(* POU D2, LD *)
FUNCTION_BLOCK D2
VAR_INPUT
	pusk: BOOL;
	KUD2: BOOL;
	RMS2_2: BOOL;
	RD2: BOOL;
	TZD2:BOOL;
	avto: BOOL;
	GRIB: BOOL;
	stop_s: BOOL;
	ruchnoe: BOOL;
	pusk_LAN: BOOL;
	stop_LAN: BOOL;
	err: BOOL;
END_VAR
VAR_OUTPUT
	ready: BOOL;
	work: BOOL;
	KM2:BOOL;
	KM3:BOOL;
	stop_D3D4: BOOL;
	avar: BOOL;
END_VAR
VAR
	prom1: BOOL;
	start_KM3: TON;
	start_KM3_prom: TON;
	KM2_prom: BOOL;
	prom: BOOL;
	tof22: TOF;
END_VAR
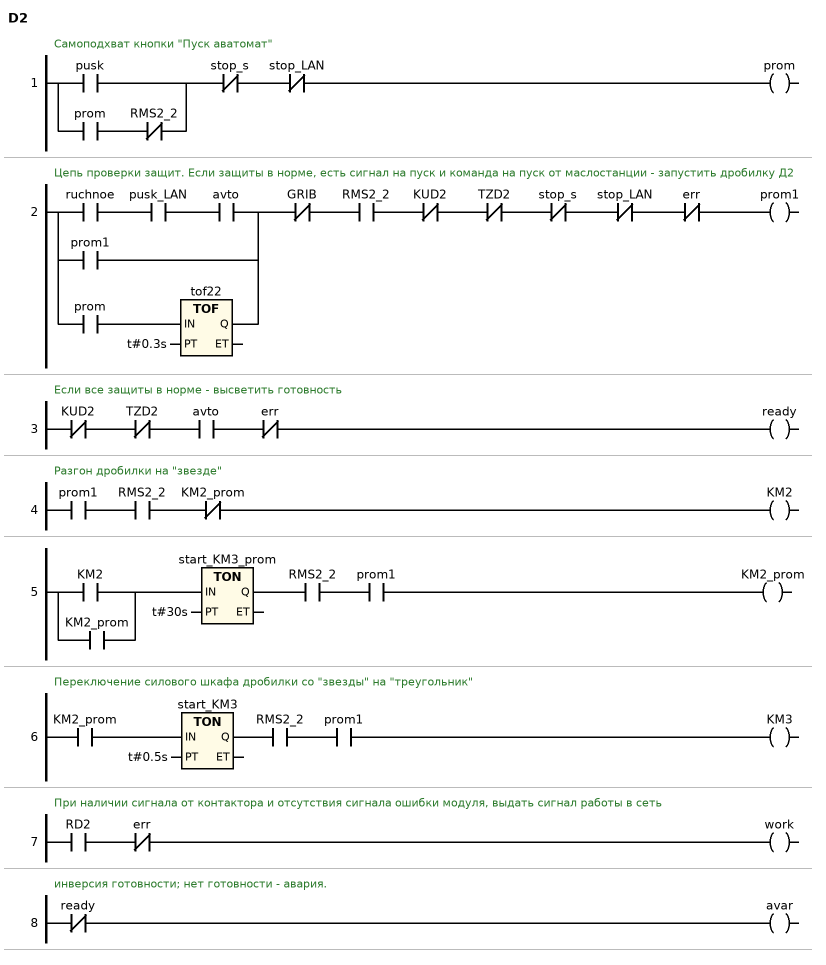
_LD_ (* Ladder Diagram *)
NETWORK 1 (* Самоподхват кнопки "Пуск аватомат" *)
	{ [pusk] | [prom] - [/RMS2_2] } - [/stop_s] - [/stop_LAN] --- (prom)
NETWORK 2 (* Цепь проверки защит. Если защиты в норме, есть сигнал на пуск и команда на пуск от маслостанции - запустить дробилку Д2 *)
	{ [ruchnoe] - [pusk_LAN] - [avto] | [prom1] | [prom] - tof22:TOF(IN: *, PT: t#0.3s) } - [/GRIB] - [RMS2_2] - [/KUD2] - [/TZD2] - [/stop_s] - [/stop_LAN] - [/err] --- (prom1)
NETWORK 3 (* Если все защиты в норме - высветить готовность *)
	[/KUD2] - [/TZD2] - [avto] - [/err] --- (ready)
NETWORK 4 (* Разгон дробилки на "звезде" *)
	[prom1] - [RMS2_2] - [/KM2_prom] --- (KM2)
NETWORK 5
	{ [KM2] | [KM2_prom] } - start_KM3_prom:TON(IN: *, PT: t#30s) - [RMS2_2] - [prom1] --- (KM2_prom)
NETWORK 6 (* Переключение силового шкафа дробилки со "звезды" на "треугольник" *)
	[KM2_prom] - start_KM3:TON(IN: *, PT: t#0.5s) - [RMS2_2] - [prom1] --- (KM3)
NETWORK 7 (* При наличии сигнала от контактора и отсутствия сигнала ошибки модуля, выдать сигнал работы в сеть *)
	[RD2] - [/err] --- (work)
NETWORK 8 (* инверсия готовности; нет готовности - авария. *)
	[/ready] --- (avar)
_END_LD_
(* the same logic as Structured Text *)
(* Network 1: Самоподхват кнопки "Пуск аватомат" *)
prom := (pusk OR prom AND NOT RMS2_2) AND NOT stop_s AND NOT stop_LAN;
(* Network 2: Цепь проверки защит. Если защиты в норме, есть сигнал на пуск и команда на пуск от маслостанции - запустить дробилку Д2 *)
tof22(IN := prom, PT := t#0.3s);
prom1 := (ruchnoe AND pusk_LAN AND avto OR prom1 OR tof22.Q) AND NOT GRIB AND RMS2_2 AND NOT KUD2 AND NOT TZD2 AND NOT stop_s AND NOT stop_LAN AND NOT err;
(* Network 3: Если все защиты в норме - высветить готовность *)
ready := NOT KUD2 AND NOT TZD2 AND avto AND NOT err;
(* Network 4: Разгон дробилки на "звезде" *)
KM2 := prom1 AND RMS2_2 AND NOT KM2_prom;
(* Network 5 *)
start_KM3_prom(IN := KM2 OR KM2_prom, PT := t#30s);
KM2_prom := start_KM3_prom.Q AND RMS2_2 AND prom1;
(* Network 6: Переключение силового шкафа дробилки со "звезды" на "треугольник" *)
start_KM3(IN := KM2_prom, PT := t#0.5s);
KM3 := start_KM3.Q AND RMS2_2 AND prom1;
(* Network 7: При наличии сигнала от контактора и отсутствия сигнала ошибки модуля, выдать сигнал работы в сеть *)
work := RD2 AND NOT err;
(* Network 8: инверсия готовности; нет готовности - авария. *)
avar := NOT ready;
END_FUNCTION_BLOCK

(* POU D3, LD *)
FUNCTION_BLOCK D3
VAR_INPUT
	pusk: BOOL;
	KU: BOOL;
	TZN: BOOL;
	KPM: BOOL;
	TZV: BOOL;

	KUD3: BOOL;
	TZD3: BOOL;
	RD3: BOOL;
	TM: WORD;
	RMS: BOOL;
	avto_in: BOOL;
	GRIB: BOOL;
	work_D2_D3: BOOL;
	stop_in: BOOL;
	ruchnoe: BOOL;
	pusk_LAN: BOOL;
	stop_LAN: BOOL;
	err: BOOL;
	UM: BOOL;
END_VAR

VAR_OUTPUT
	KM1: BOOL;
	KM2: BOOL;
	KM3: BOOL;
	ready: BOOL;
	nasos: BOOL;
	vent: BOOL;
	ten: BOOL;
	work: BOOL;
	avto:BOOL;
	avar: BOOL;
	stop_D3D4: BOOL;
	tm_ins: BOOL;
END_VAR

VAR
	prom1: BOOL;
	start_KM3: TON;
	KM2_prom: BOOL;
	start_KM3_prom: TON;
	run_pump: TON;
	prom2: BOOL;
	stop_D4: TON;
	stop_pump: TOF;
	tm_vent_ins: BOOL;
	tof1: TOF;
END_VAR
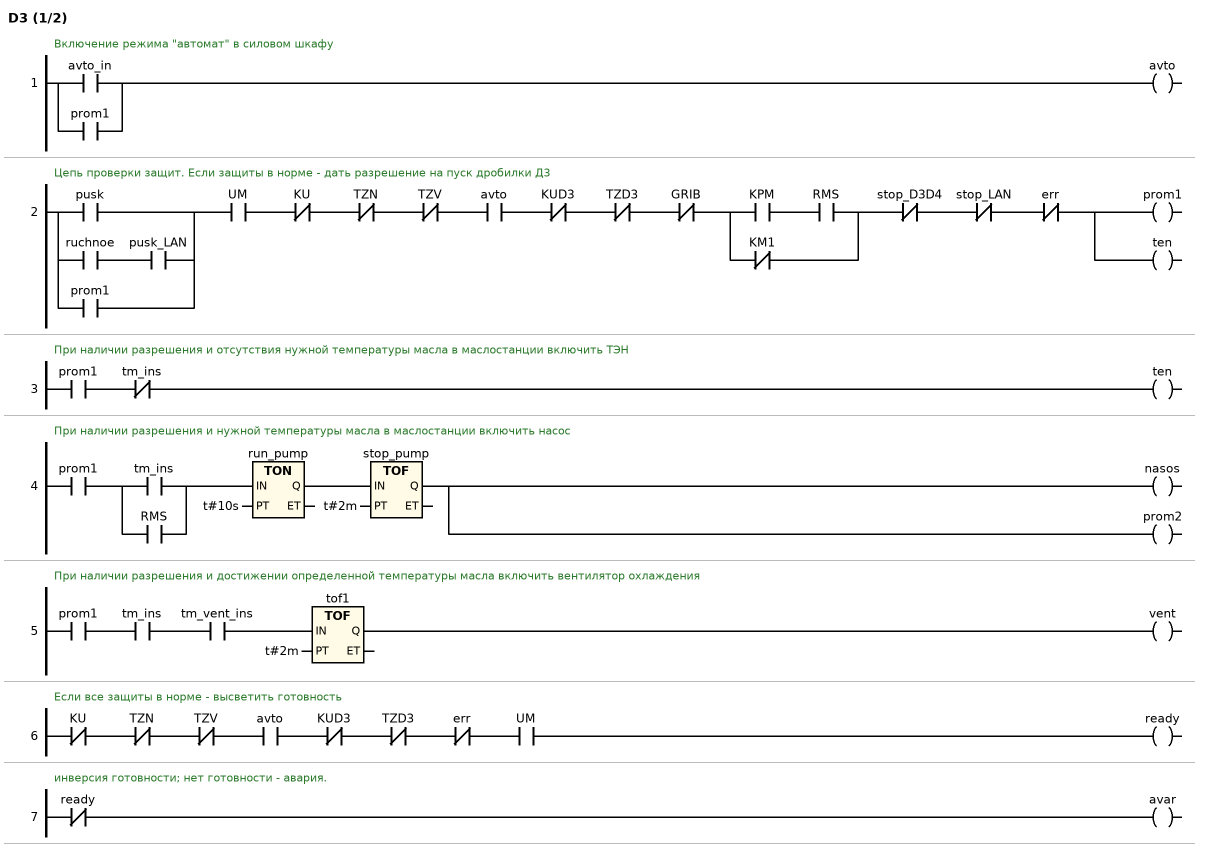
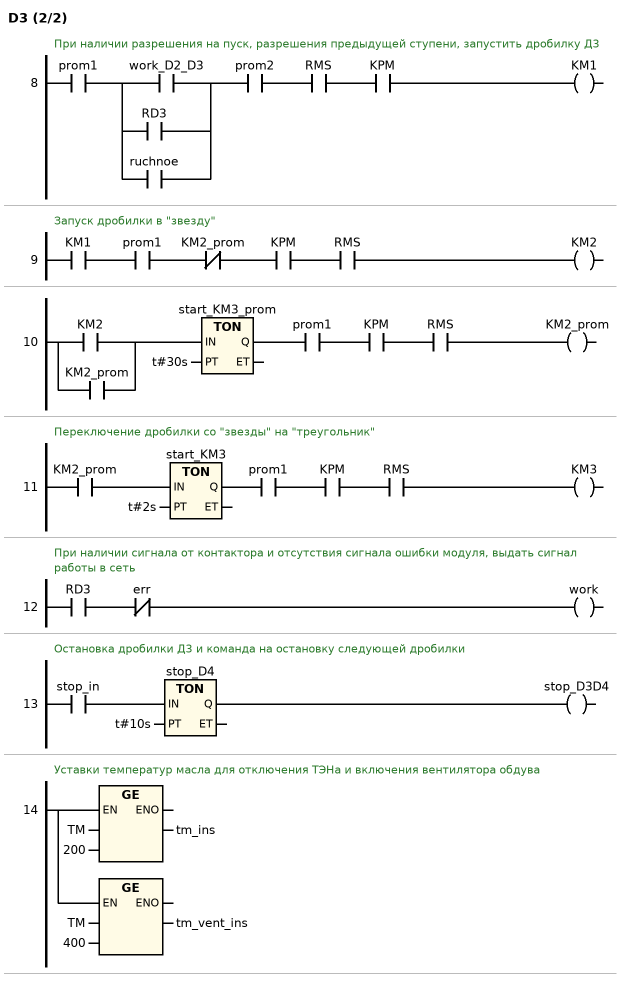
_LD_ (* Ladder Diagram *)
NETWORK 1 (* Включение режима "автомат" в силовом шкафу *)
	{ [avto_in] | [prom1] } --- (avto)
NETWORK 2 (* Цепь проверки защит. Если защиты в норме - дать разрешение на пуск дробилки Д3 *)
	{ [pusk] | [ruchnoe] - [pusk_LAN] | [prom1] } - [UM] - [/KU] - [/TZN] - [/TZV] - [avto] - [/KUD3] - [/TZD3] - [/GRIB] - { [KPM] - [RMS] | [/KM1] } - [/stop_D3D4] - [/stop_LAN] - [/err] --- (prom1) (ten)
NETWORK 3 (* При наличии разрешения и отсутствия нужной температуры масла в маслостанции включить ТЭН *)
	[prom1] - [/tm_ins] --- (ten)
NETWORK 4 (* При наличии разрешения и нужной температуры масла в маслостанции включить насос *)
	[prom1] - { [tm_ins] | [RMS] } - run_pump:TON(IN: *, PT: t#10s) - stop_pump:TOF(IN: *, PT: t#2m) --- (nasos) (prom2)
NETWORK 5 (* При наличии разрешения и достижении определенной температуры масла включить вентилятор охлаждения *)
	[prom1] - [tm_ins] - [tm_vent_ins] - tof1:TOF(IN: *, PT: t#2m) --- (vent)
NETWORK 6 (* Если все защиты в норме - высветить готовность *)
	[/KU] - [/TZN] - [/TZV] - [avto] - [/KUD3] - [/TZD3] - [/err] - [UM] --- (ready)
NETWORK 7 (* инверсия готовности; нет готовности - авария. *)
	[/ready] --- (avar)
NETWORK 8 (* При наличии разрешения на пуск, разрешения предыдущей ступени, запустить дробилку Д3 *)
	[prom1] - { [work_D2_D3] | [RD3] | [ruchnoe] } - [prom2] - [RMS] - [KPM] --- (KM1)
NETWORK 9 (* Запуск дробилки в "звезду" *)
	[KM1] - [prom1] - [/KM2_prom] - [KPM] - [RMS] --- (KM2)
NETWORK 10
	{ [KM2] | [KM2_prom] } - start_KM3_prom:TON(IN: *, PT: t#30s) - [prom1] - [KPM] - [RMS] --- (KM2_prom)
NETWORK 11 (* Переключение дробилки со "звезды" на "треугольник" *)
	[KM2_prom] - start_KM3:TON(IN: *, PT: t#2s) - [prom1] - [KPM] - [RMS] --- (KM3)
NETWORK 12 (* При наличии сигнала от контактора и отсутствия сигнала ошибки модуля, выдать сигнал работы в сеть *)
	[RD3] - [/err] --- (work)
NETWORK 13 (* Остановка дробилки Д3 и команда на остановку следующей дробилки *)
	[stop_in] - stop_D4:TON(IN: *, PT: t#10s) --- (stop_D3D4)
NETWORK 14 (* Уставки температур масла для отключения ТЭНа и включения вентилятора обдува *)
	*
		EN --- GE(TM, 200) => tm_ins
		EN --- GE(TM, 400) => tm_vent_ins
_END_LD_
(* the same logic as Structured Text *)
(* Network 1: Включение режима "автомат" в силовом шкафу *)
avto := avto_in OR prom1;
(* Network 2: Цепь проверки защит. Если защиты в норме - дать разрешение на пуск дробилки Д3 *)
prom1 := (pusk OR ruchnoe AND pusk_LAN OR prom1) AND UM AND NOT KU AND NOT TZN AND NOT TZV AND avto AND NOT KUD3 AND NOT TZD3 AND NOT GRIB AND (KPM AND RMS OR NOT KM1) AND NOT stop_D3D4 AND NOT stop_LAN AND NOT err;
ten := prom1;
(* Network 3: При наличии разрешения и отсутствия нужной температуры масла в маслостанции включить ТЭН *)
ten := prom1 AND NOT tm_ins;
(* Network 4: При наличии разрешения и нужной температуры масла в маслостанции включить насос *)
run_pump(IN := prom1 AND (tm_ins OR RMS), PT := t#10s);
stop_pump(IN := run_pump.Q, PT := t#2m);
nasos := stop_pump.Q;
prom2 := stop_pump.Q;
(* Network 5: При наличии разрешения и достижении определенной температуры масла включить вентилятор охлаждения *)
tof1(IN := prom1 AND tm_ins AND tm_vent_ins, PT := t#2m);
vent := tof1.Q;
(* Network 6: Если все защиты в норме - высветить готовность *)
ready := NOT KU AND NOT TZN AND NOT TZV AND avto AND NOT KUD3 AND NOT TZD3 AND NOT err AND UM;
(* Network 7: инверсия готовности; нет готовности - авария. *)
avar := NOT ready;
(* Network 8: При наличии разрешения на пуск, разрешения предыдущей ступени, запустить дробилку Д3 *)
KM1 := prom1 AND (work_D2_D3 OR RD3 OR ruchnoe) AND prom2 AND RMS AND KPM;
(* Network 9: Запуск дробилки в "звезду" *)
KM2 := KM1 AND prom1 AND NOT KM2_prom AND KPM AND RMS;
(* Network 10 *)
start_KM3_prom(IN := KM2 OR KM2_prom, PT := t#30s);
KM2_prom := start_KM3_prom.Q AND prom1 AND KPM AND RMS;
(* Network 11: Переключение дробилки со "звезды" на "треугольник" *)
start_KM3(IN := KM2_prom, PT := t#2s);
KM3 := start_KM3.Q AND prom1 AND KPM AND RMS;
(* Network 12: При наличии сигнала от контактора и отсутствия сигнала ошибки модуля, выдать сигнал работы в сеть *)
work := RD3 AND NOT err;
(* Network 13: Остановка дробилки Д3 и команда на остановку следующей дробилки *)
stop_D4(IN := stop_in, PT := t#10s);
stop_D3D4 := stop_D4.Q;
(* Network 14: Уставки температур масла для отключения ТЭНа и включения вентилятора обдува *)
tm_ins := TM >= 200;
tm_vent_ins := TM >= 400;
END_FUNCTION_BLOCK

(* POU D4, LD *)
FUNCTION_BLOCK D4
VAR_INPUT
	pusk: BOOL;
	KU: BOOL;
	TZN: BOOL;
	KPM: BOOL;
	TZV: BOOL;

	KUD3: BOOL;
	TZD3: BOOL;
	RD3: BOOL;
	TM: WORD;
	RMS: BOOL;
	avto_in: BOOL;
	GRIB: BOOL;
	work_D2_D3: BOOL;
	stop_in: BOOL;
	ruchnoe: BOOL;
	ins_0_40: BOOL;
	pusk_LAN: BOOL;
	stop_LAN: BOOL;
	err: BOOL;
	UM: BOOL;
END_VAR

VAR_OUTPUT
	KM1: BOOL;
	KM2: BOOL;
	KM3: BOOL;
	ready: BOOL;
	nasos: BOOL;
	vent: BOOL;
	ten: BOOL;
	work: BOOL;
	avto:BOOL;
	avar: BOOL;
	stop_D3D4: BOOL;
	tm_ins: BOOL;
END_VAR

VAR
	prom1: BOOL;
	start_KM3: TON;
	KM2_prom: BOOL;
	start_KM3_prom: TON;
	run_pump: TON;
	prom2: BOOL;
	stop_D4: TON;
	stop_pump: TOF;
	tm_vent_ins: BOOL;
	tof1: TOF;
END_VAR
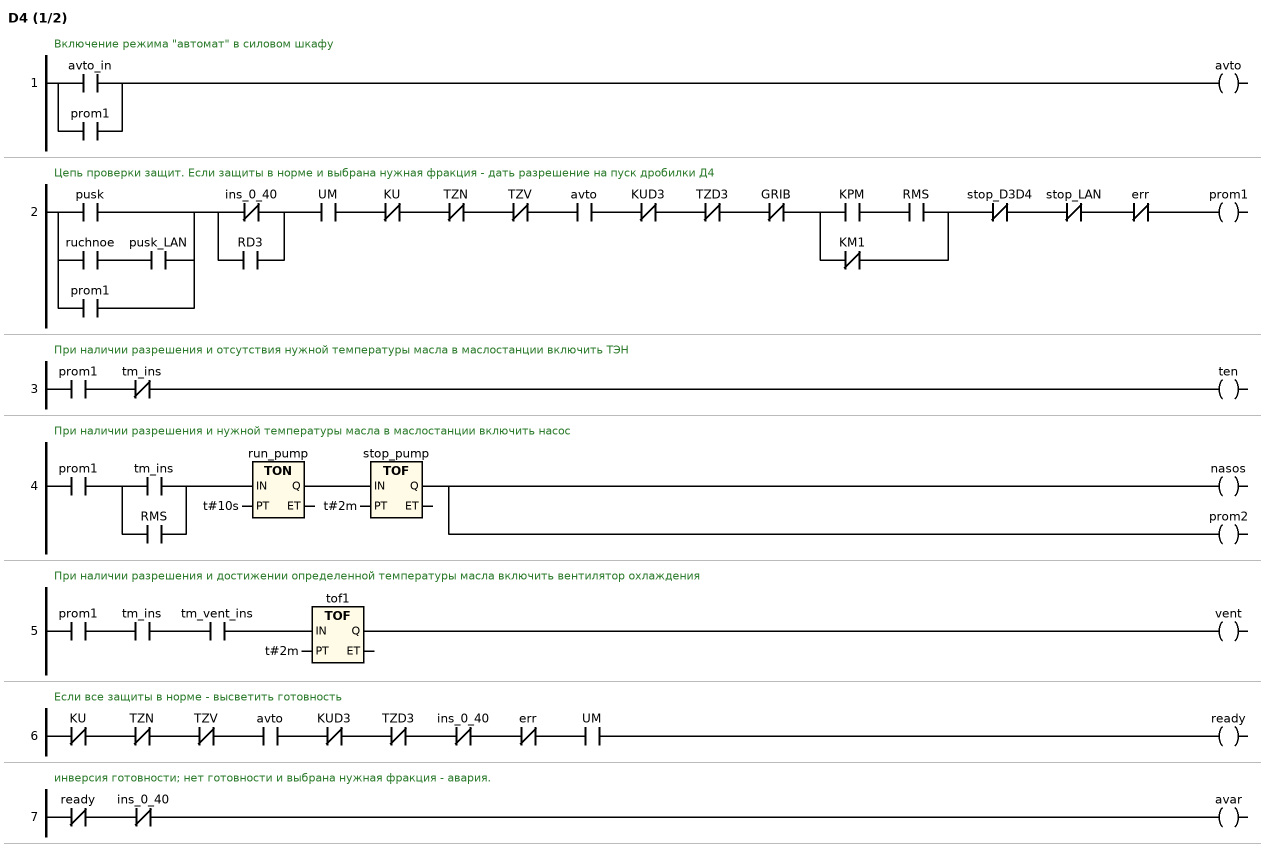
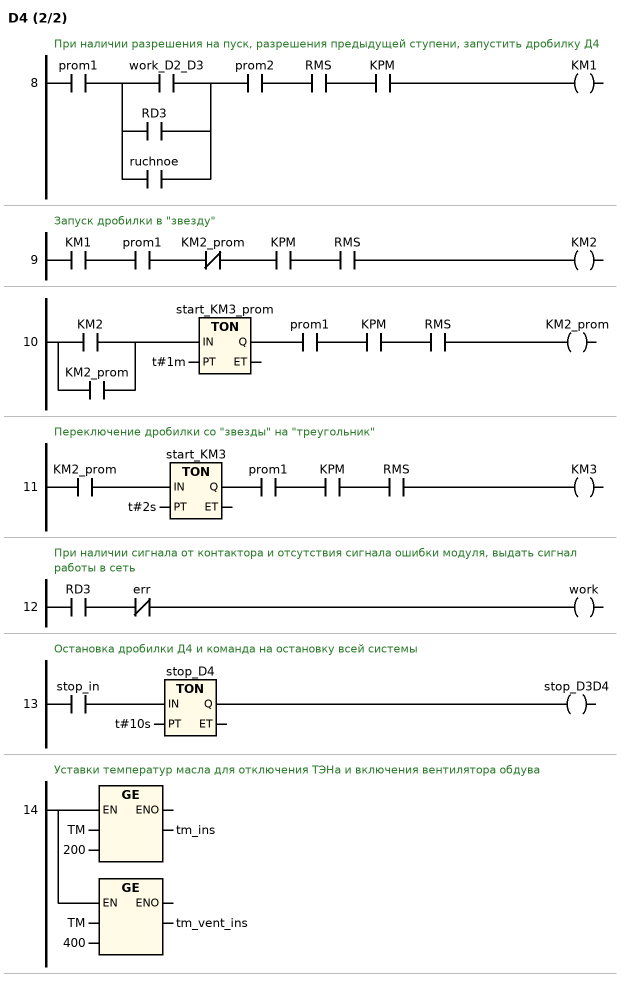
_LD_ (* Ladder Diagram *)
NETWORK 1 (* Включение режима "автомат" в силовом шкафу *)
	{ [avto_in] | [prom1] } --- (avto)
NETWORK 2 (* Цепь проверки защит. Если защиты в норме и выбрана нужная фракция - дать разрешение на пуск дробилки Д4 *)
	{ [pusk] | [ruchnoe] - [pusk_LAN] | [prom1] } - { [/ins_0_40] | [RD3] } - [UM] - [/KU] - [/TZN] - [/TZV] - [avto] - [/KUD3] - [/TZD3] - [/GRIB] - { [KPM] - [RMS] | [/KM1] } - [/stop_D3D4] - [/stop_LAN] - [/err] --- (prom1)
NETWORK 3 (* При наличии разрешения и отсутствия нужной температуры масла в маслостанции включить ТЭН *)
	[prom1] - [/tm_ins] --- (ten)
NETWORK 4 (* При наличии разрешения и нужной температуры масла в маслостанции включить насос *)
	[prom1] - { [tm_ins] | [RMS] } - run_pump:TON(IN: *, PT: t#10s) - stop_pump:TOF(IN: *, PT: t#2m) --- (nasos) (prom2)
NETWORK 5 (* При наличии разрешения и достижении определенной температуры масла включить вентилятор охлаждения *)
	[prom1] - [tm_ins] - [tm_vent_ins] - tof1:TOF(IN: *, PT: t#2m) --- (vent)
NETWORK 6 (* Если все защиты в норме - высветить готовность *)
	[/KU] - [/TZN] - [/TZV] - [avto] - [/KUD3] - [/TZD3] - [/ins_0_40] - [/err] - [UM] --- (ready)
NETWORK 7 (* инверсия готовности; нет готовности и выбрана нужная фракция - авария. *)
	[/ready] - [/ins_0_40] --- (avar)
NETWORK 8 (* При наличии разрешения на пуск, разрешения предыдущей ступени, запустить дробилку Д4 *)
	[prom1] - { [work_D2_D3] | [RD3] | [ruchnoe] } - [prom2] - [RMS] - [KPM] --- (KM1)
NETWORK 9 (* Запуск дробилки в "звезду" *)
	[KM1] - [prom1] - [/KM2_prom] - [KPM] - [RMS] --- (KM2)
NETWORK 10
	{ [KM2] | [KM2_prom] } - start_KM3_prom:TON(IN: *, PT: t#1m) - [prom1] - [KPM] - [RMS] --- (KM2_prom)
NETWORK 11 (* Переключение дробилки со "звезды" на "треугольник" *)
	[KM2_prom] - start_KM3:TON(IN: *, PT: t#2s) - [prom1] - [KPM] - [RMS] --- (KM3)
NETWORK 12 (* При наличии сигнала от контактора и отсутствия сигнала ошибки модуля, выдать сигнал работы в сеть *)
	[RD3] - [/err] --- (work)
NETWORK 13 (* Остановка дробилки Д4 и команда на остановку всей системы *)
	[stop_in] - stop_D4:TON(IN: *, PT: t#10s) --- (stop_D3D4)
NETWORK 14 (* Уставки температур масла для отключения ТЭНа и включения вентилятора обдува *)
	*
		EN --- GE(TM, 200) => tm_ins
		EN --- GE(TM, 400) => tm_vent_ins
_END_LD_
(* the same logic as Structured Text *)
(* Network 1: Включение режима "автомат" в силовом шкафу *)
avto := avto_in OR prom1;
(* Network 2: Цепь проверки защит. Если защиты в норме и выбрана нужная фракция - дать разрешение на пуск дробилки Д4 *)
prom1 := (pusk OR ruchnoe AND pusk_LAN OR prom1) AND (NOT ins_0_40 OR RD3) AND UM AND NOT KU AND NOT TZN AND NOT TZV AND avto AND NOT KUD3 AND NOT TZD3 AND NOT GRIB AND (KPM AND RMS OR NOT KM1) AND NOT stop_D3D4 AND NOT stop_LAN AND NOT err;
(* Network 3: При наличии разрешения и отсутствия нужной температуры масла в маслостанции включить ТЭН *)
ten := prom1 AND NOT tm_ins;
(* Network 4: При наличии разрешения и нужной температуры масла в маслостанции включить насос *)
run_pump(IN := prom1 AND (tm_ins OR RMS), PT := t#10s);
stop_pump(IN := run_pump.Q, PT := t#2m);
nasos := stop_pump.Q;
prom2 := stop_pump.Q;
(* Network 5: При наличии разрешения и достижении определенной температуры масла включить вентилятор охлаждения *)
tof1(IN := prom1 AND tm_ins AND tm_vent_ins, PT := t#2m);
vent := tof1.Q;
(* Network 6: Если все защиты в норме - высветить готовность *)
ready := NOT KU AND NOT TZN AND NOT TZV AND avto AND NOT KUD3 AND NOT TZD3 AND NOT ins_0_40 AND NOT err AND UM;
(* Network 7: инверсия готовности; нет готовности и выбрана нужная фракция - авария. *)
avar := NOT ready AND NOT ins_0_40;
(* Network 8: При наличии разрешения на пуск, разрешения предыдущей ступени, запустить дробилку Д4 *)
KM1 := prom1 AND (work_D2_D3 OR RD3 OR ruchnoe) AND prom2 AND RMS AND KPM;
(* Network 9: Запуск дробилки в "звезду" *)
KM2 := KM1 AND prom1 AND NOT KM2_prom AND KPM AND RMS;
(* Network 10 *)
start_KM3_prom(IN := KM2 OR KM2_prom, PT := t#1m);
KM2_prom := start_KM3_prom.Q AND prom1 AND KPM AND RMS;
(* Network 11: Переключение дробилки со "звезды" на "треугольник" *)
start_KM3(IN := KM2_prom, PT := t#2s);
KM3 := start_KM3.Q AND prom1 AND KPM AND RMS;
(* Network 12: При наличии сигнала от контактора и отсутствия сигнала ошибки модуля, выдать сигнал работы в сеть *)
work := RD3 AND NOT err;
(* Network 13: Остановка дробилки Д4 и команда на остановку всей системы *)
stop_D4(IN := stop_in, PT := t#10s);
stop_D3D4 := stop_D4.Q;
(* Network 14: Уставки температур масла для отключения ТЭНа и включения вентилятора обдува *)
tm_ins := TM >= 200;
tm_vent_ins := TM >= 400;
END_FUNCTION_BLOCK

(* POU LK1, LD *)
FUNCTION_BLOCK LK1 (*функциональный блок управления ленточными конвеерами 3, 5, 7, 8, 10-13*)
VAR_INPUT
	pusk: BOOL;
	avto:BOOL;
	KU: BOOL;
	TZ: BOOL;
	tros: BOOL;
	shod: BOOL;
	ogr: BOOL;
	VL:BOOL;
	P: BOOL;
	GRIB: BOOL;
	stop_s: BOOL;
	ruchnoe: BOOL;
	pusk_LAN: BOOL;
	stop_LAN: BOOL;
	err: BOOL;
	tros_self: BOOL;
	shod_self: BOOL;
	ogr_self: BOOL;
	pusk_sys_ins:BOOL;
END_VAR

VAR_OUTPUT
	KM:BOOL;
	ready: BOOL;
	work: BOOL;
	avar: BOOL;
	avar_vl: BOOL;
END_VAR

VAR
	prom1: BOOL;

	ftrig: F_TRIG;
	SR: SR;
END_VAR
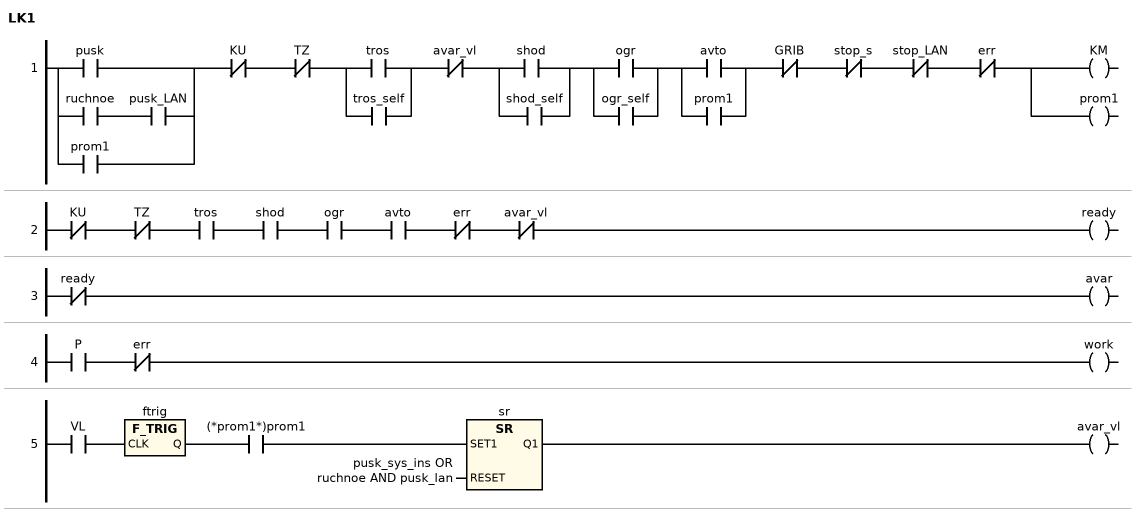
_LD_ (* Ladder Diagram *)
NETWORK 1
	{ [pusk] | [ruchnoe] - [pusk_LAN] | [prom1] } - [/KU] - [/TZ] - { [tros] | [tros_self] } - [/avar_vl] - { [shod] | [shod_self] } - { [ogr] | [ogr_self] } - { [avto] | [prom1] } - [/GRIB] - [/stop_s] - [/stop_LAN] - [/err] --- (KM) (prom1)
NETWORK 2
	[/KU] - [/TZ] - [tros] - [shod] - [ogr] - [avto] - [/err] - [/avar_vl] --- (ready)
NETWORK 3
	[/ready] --- (avar)
NETWORK 4
	[P] - [/err] --- (work)
NETWORK 5
	[VL] - ftrig:F_TRIG(CLK: *) - [(*prom1*)prom1] - sr:SR(SET1: *, RESET: pusk_sys_ins OR ruchnoe AND pusk_lan) --- (avar_vl)
_END_LD_
(* the same logic as Structured Text *)
(* Network 1 *)
KM := (pusk OR ruchnoe AND pusk_LAN OR prom1) AND NOT KU AND NOT TZ AND (tros OR tros_self) AND NOT avar_vl AND (shod OR shod_self) AND (ogr OR ogr_self) AND (avto OR prom1) AND NOT GRIB AND NOT stop_s AND NOT stop_LAN AND NOT err;
prom1 := KM;
(* Network 2 *)
ready := NOT KU AND NOT TZ AND tros AND shod AND ogr AND avto AND NOT err AND NOT avar_vl;
(* Network 3 *)
avar := NOT ready;
(* Network 4 *)
work := P AND NOT err;
(* Network 5 *)
ftrig(CLK := VL);
sr(SET1 := ftrig.Q AND ((*prom1*)prom1), RESET := pusk_sys_ins OR ruchnoe AND pusk_lan);
avar_vl := sr.Q1;
END_FUNCTION_BLOCK

(* POU counter, LD *)
FUNCTION_BLOCK counter  (* блок косвенного подсчёта скорости, исходя из приходящего количества импульсов*)
VAR_INPUT
	Vl: WORD;
	work: BOOL;
	in_time: WORD;
END_VAR
VAR_OUTPUT
	out_Vl: BOOL;
END_VAR
VAR
	vl_ins: WORD;
	vl_eq: BOOL;
	ton1: TOF;
	blink1: BLINK;
	tp1: TP;
	vl_sub: WORD;
	ins_time: WORD;
	time_read: TIME;
END_VAR
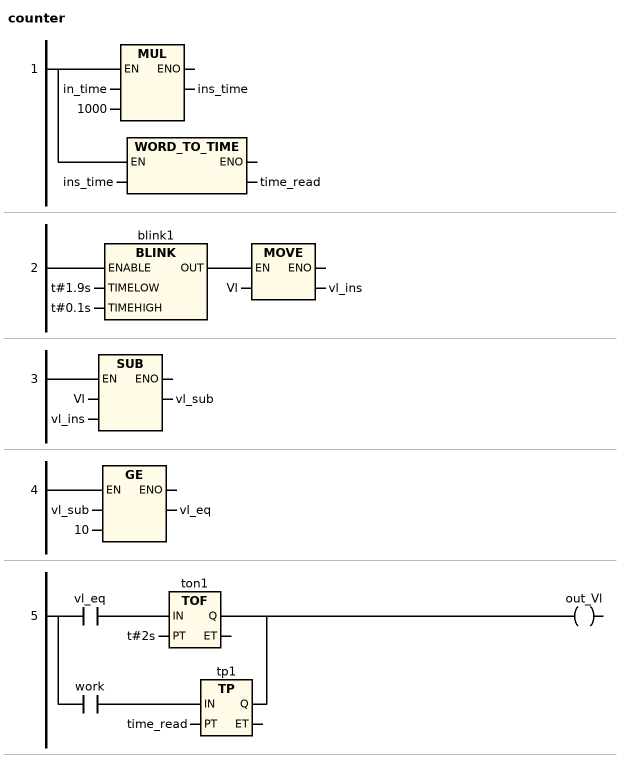
_LD_ (* Ladder Diagram *)
NETWORK 1
	*
		EN --- MUL(in_time, 1000) => ins_time
		EN --- WORD_TO_TIME(ins_time) => time_read
NETWORK 2
	blink1:BLINK(ENABLE: *, TIMELOW: t#1.9s, TIMEHIGH: t#0.1s)
		EN --- MOVE(Vl) => vl_ins
NETWORK 3
	*
		EN --- SUB(Vl, vl_ins) => vl_sub
NETWORK 4
	*
		EN --- GE(vl_sub, 10) => vl_eq
NETWORK 5
	{ [vl_eq] - ton1:TOF(IN: *, PT: t#2s) | [work] - tp1:TP(IN: *, PT: time_read) } --- (out_Vl)
_END_LD_
(* the same logic as Structured Text *)
(* Network 1 *)
ins_time := in_time * 1000;
time_read := WORD_TO_TIME(ins_time);
(* Network 2 *)
blink1(ENABLE := TRUE, TIMELOW := t#1.9s, TIMEHIGH := t#0.1s);
IF blink1.OUT THEN
	vl_ins := Vl;
END_IF;
(* Network 3 *)
vl_sub := Vl - vl_ins;
(* Network 4 *)
vl_eq := vl_sub >= 10;
(* Network 5 *)
ton1(IN := vl_eq, PT := t#2s);
tp1(IN := work, PT := time_read);
out_Vl := ton1.Q OR tp1.Q;
END_FUNCTION_BLOCK

(* POU LK12, LD *)
FUNCTION_BLOCK LK12 (*функциональный блок управления ленточными конвеерами 3, 5, 7, 8, 10-13*)
VAR_INPUT
	avto:BOOL;
	KU: BOOL;
	TZ: BOOL;
	tros: BOOL;
	shod: BOOL;
	ogr: BOOL;
	VL:BOOL;
	P: BOOL;
	GRIB: BOOL;
	stop_s: BOOL;
	ruchnoe: BOOL;
	pusk_LAN: BOOL;
	stop_LAN: BOOL;
	err: BOOL;
	tros_self: BOOL;
	shod_self: BOOL;
	ogr_self: BOOL;
	pusk_sys_ins:BOOL;
END_VAR

VAR_OUTPUT
	KM:BOOL;
	ready: BOOL;
	work: BOOL;
	avar: BOOL;
	avar_vl: BOOL;
END_VAR

VAR
	prom1: BOOL;

	ftrig: F_TRIG;
	SR: SR;
END_VAR
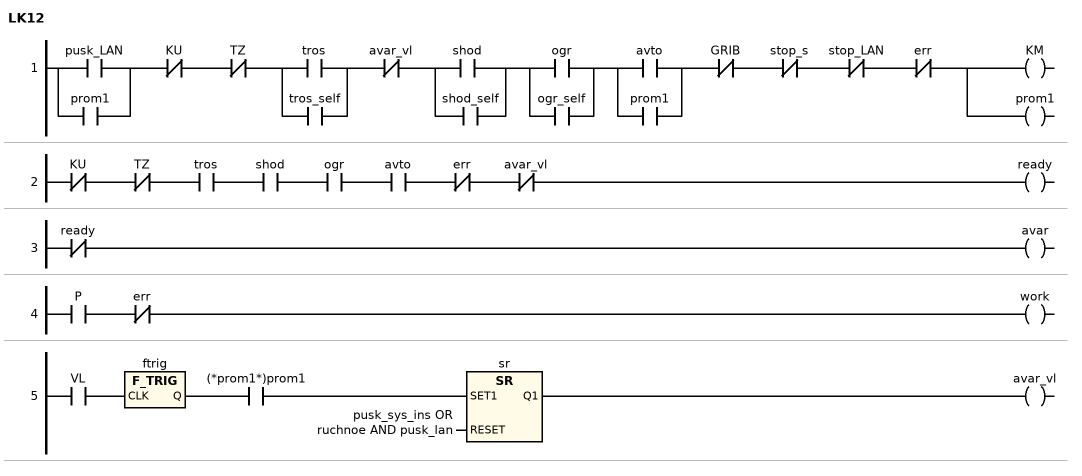
_LD_ (* Ladder Diagram *)
NETWORK 1
	{ [pusk_LAN] | [prom1] } - [/KU] - [/TZ] - { [tros] | [tros_self] } - [/avar_vl] - { [shod] | [shod_self] } - { [ogr] | [ogr_self] } - { [avto] | [prom1] } - [/GRIB] - [/stop_s] - [/stop_LAN] - [/err] --- (KM) (prom1)
NETWORK 2
	[/KU] - [/TZ] - [tros] - [shod] - [ogr] - [avto] - [/err] - [/avar_vl] --- (ready)
NETWORK 3
	[/ready] --- (avar)
NETWORK 4
	[P] - [/err] --- (work)
NETWORK 5
	[VL] - ftrig:F_TRIG(CLK: *) - [(*prom1*)prom1] - sr:SR(SET1: *, RESET: pusk_sys_ins OR ruchnoe AND pusk_lan) --- (avar_vl)
_END_LD_
(* the same logic as Structured Text *)
(* Network 1 *)
KM := (pusk_LAN OR prom1) AND NOT KU AND NOT TZ AND (tros OR tros_self) AND NOT avar_vl AND (shod OR shod_self) AND (ogr OR ogr_self) AND (avto OR prom1) AND NOT GRIB AND NOT stop_s AND NOT stop_LAN AND NOT err;
prom1 := KM;
(* Network 2 *)
ready := NOT KU AND NOT TZ AND tros AND shod AND ogr AND avto AND NOT err AND NOT avar_vl;
(* Network 3 *)
avar := NOT ready;
(* Network 4 *)
work := P AND NOT err;
(* Network 5 *)
ftrig(CLK := VL);
sr(SET1 := ftrig.Q AND ((*prom1*)prom1), RESET := pusk_sys_ins OR ruchnoe AND pusk_lan);
avar_vl := sr.Q1;
END_FUNCTION_BLOCK

(* POU LK12_modern, LD *)
FUNCTION_BLOCK LK12_modern (*функциональный блок управления ленточными конвеерами 12*)
VAR_INPUT
	pusk: BOOL;
	avto:BOOL;
	KU: BOOL;
	TZ: BOOL;
	tros: BOOL;
	shod: BOOL;
	ogr: BOOL;
	VL:BOOL;
	P: BOOL;
	GRIB: BOOL;
	stop_s: BOOL;
	ruchnoe: BOOL;
	pusk_LAN: BOOL;
	stop_LAN: BOOL;
	err: BOOL;
	tros_self: BOOL;
	shod_self: BOOL;
	ogr_self: BOOL;
	pusk_sys_ins:BOOL;
	switcher_in: WORD;
	current_value_lk12_in: BOOL;
END_VAR

VAR_OUTPUT
	KM:BOOL;
	ready: BOOL;
	work: BOOL;
	avar: BOOL;
	avar_vl: BOOL;
	current_value_lk12_out: BOOL;
END_VAR

VAR
	prom1: BOOL;

	ftrig: F_TRIG;
	SR: SR;
	switcher_in_bool: BOOL;
	lk12_trig: lk12_trig;
END_VAR
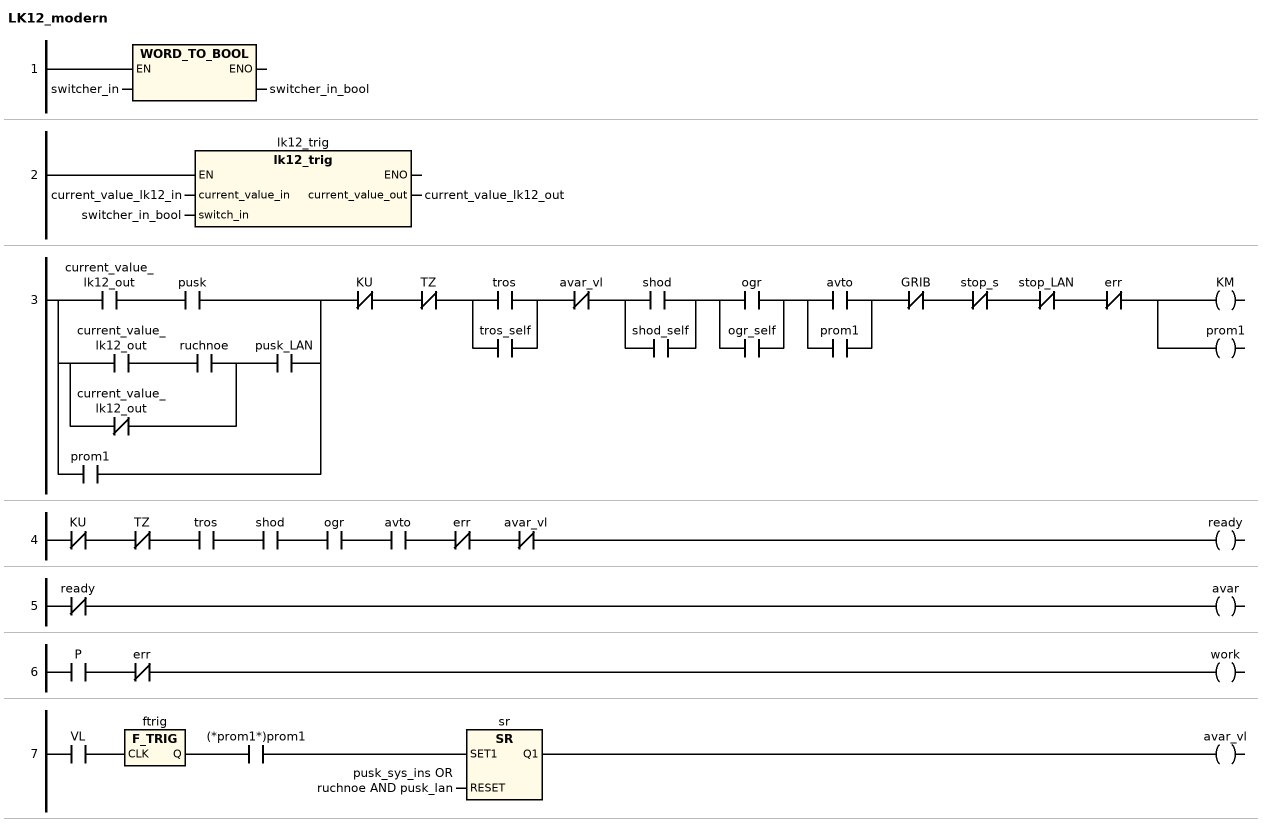
_LD_ (* Ladder Diagram *)
NETWORK 1
	*
		EN --- WORD_TO_BOOL(switcher_in) => switcher_in_bool
NETWORK 2
	*
		EN --- lk12_trig:lk12_trig(current_value_in: current_value_lk12_in, switch_in: switcher_in_bool) => current_value_lk12_out
NETWORK 3
	{ [current_value_lk12_out] - [pusk] | { [current_value_lk12_out] - [ruchnoe] | [/current_value_lk12_out] } - [pusk_LAN] | [prom1] } - [/KU] - [/TZ] - { [tros] | [tros_self] } - [/avar_vl] - { [shod] | [shod_self] } - { [ogr] | [ogr_self] } - { [avto] | [prom1] } - [/GRIB] - [/stop_s] - [/stop_LAN] - [/err] --- (KM) (prom1)
NETWORK 4
	[/KU] - [/TZ] - [tros] - [shod] - [ogr] - [avto] - [/err] - [/avar_vl] --- (ready)
NETWORK 5
	[/ready] --- (avar)
NETWORK 6
	[P] - [/err] --- (work)
NETWORK 7
	[VL] - ftrig:F_TRIG(CLK: *) - [(*prom1*)prom1] - sr:SR(SET1: *, RESET: pusk_sys_ins OR ruchnoe AND pusk_lan) --- (avar_vl)
_END_LD_
(* the same logic as Structured Text *)
(* Network 1 *)
switcher_in_bool := WORD_TO_BOOL(switcher_in);
(* Network 2 *)
lk12_trig(current_value_in := current_value_lk12_in, switch_in := switcher_in_bool);
current_value_lk12_out := lk12_trig.current_value_out;
(* Network 3 *)
KM := (current_value_lk12_out AND pusk OR (current_value_lk12_out AND ruchnoe OR NOT current_value_lk12_out) AND pusk_LAN OR prom1) AND NOT KU AND NOT TZ AND (tros OR tros_self) AND NOT avar_vl AND (shod OR shod_self) AND (ogr OR ogr_self) AND (avto OR prom1) AND NOT GRIB AND NOT stop_s AND NOT stop_LAN AND NOT err;
prom1 := KM;
(* Network 4 *)
ready := NOT KU AND NOT TZ AND tros AND shod AND ogr AND avto AND NOT err AND NOT avar_vl;
(* Network 5 *)
avar := NOT ready;
(* Network 6 *)
work := P AND NOT err;
(* Network 7 *)
ftrig(CLK := VL);
sr(SET1 := ftrig.Q AND ((*prom1*)prom1), RESET := pusk_sys_ins OR ruchnoe AND pusk_lan);
avar_vl := sr.Q1;
END_FUNCTION_BLOCK

(* POU lk12_trig, ST *)
FUNCTION_BLOCK lk12_trig
VAR_INPUT
	current_value_in: BOOL;
	switch_in: BOOL;
END_VAR
VAR_OUTPUT
	current_value_out: BOOL;
END_VAR
VAR
	rtrig : R_TRIG;
	rtrigQ: BOOL;
END_VAR
rtrig(CLK := switch_in);
rtrigQ := rtrig.Q;

IF current_value_in = TRUE AND rtrigQ = TRUE
THEN
current_value_out := FALSE;
ELSIF current_value_in = FALSE AND rtrigQ = TRUE
THEN
current_value_out := TRUE;
END_IF
END_FUNCTION_BLOCK

(* POU Grohot, LD *)
FUNCTION_BLOCK Grohot
VAR_INPUT
	pusk: BOOL;
	avto: BOOL;
	KU: BOOL;
	TZ: BOOL;
	P:BOOL;
	STOP: BOOL;
	GRIB: BOOL;
	stop_s: BOOL;
	ruchnoe: BOOL;
	pusk_LAN: BOOL;
	stop_LAN: BOOL;
	err: BOOL;
END_VAR

VAR_OUTPUT
	KM: BOOL;
	ready: BOOL;
	work: BOOL;
	avar: BOOL;
END_VAR

VAR
	prom1: BOOL;
END_VAR
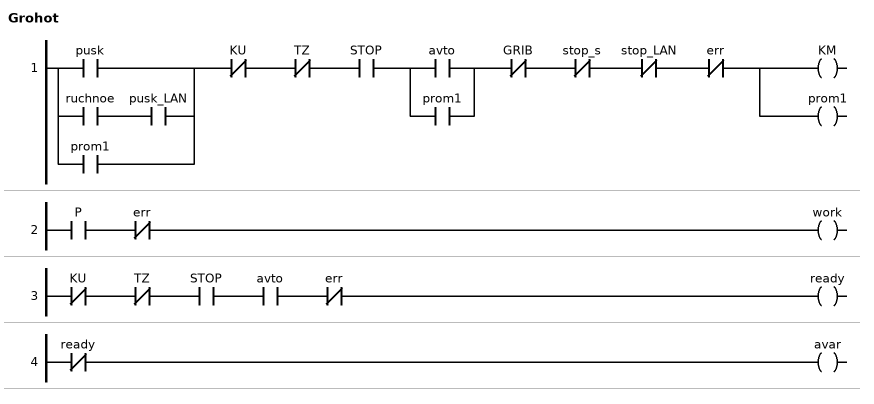
_LD_ (* Ladder Diagram *)
NETWORK 1
	{ [pusk] | [ruchnoe] - [pusk_LAN] | [prom1] } - [/KU] - [/TZ] - [STOP] - { [avto] | [prom1] } - [/GRIB] - [/stop_s] - [/stop_LAN] - [/err] --- (KM) (prom1)
NETWORK 2
	[P] - [/err] --- (work)
NETWORK 3
	[/KU] - [/TZ] - [STOP] - [avto] - [/err] --- (ready)
NETWORK 4
	[/ready] --- (avar)
_END_LD_
(* the same logic as Structured Text *)
(* Network 1 *)
KM := (pusk OR ruchnoe AND pusk_LAN OR prom1) AND NOT KU AND NOT TZ AND STOP AND (avto OR prom1) AND NOT GRIB AND NOT stop_s AND NOT stop_LAN AND NOT err;
prom1 := KM;
(* Network 2 *)
work := P AND NOT err;
(* Network 3 *)
ready := NOT KU AND NOT TZ AND STOP AND avto AND NOT err;
(* Network 4 *)
avar := NOT ready;
END_FUNCTION_BLOCK

(* POU LK3, LD *)
FUNCTION_BLOCK LK3  (*Ленточный конвееры 6*)
VAR_INPUT
	pusk: BOOL;
	avto:BOOL;
	KU: BOOL;
	TZ: BOOL;
	tros: BOOL;
	shod: BOOL;
	ogr: BOOL;
	VL:BOOL;
	P:BOOL;
	in_020: BOOL;
	stop_s: BOOL;
	GRIB: BOOL;
	ruchnoe: BOOL;
	pusk_LAN: BOOL;
	stop_LAN: BOOL;
	err: BOOL;
	tros_self: BOOL;
	shod_self: BOOL;
	ogr_self: BOOL;
	pusk_sys_ins:BOOL;
END_VAR

VAR_OUTPUT
	KM: BOOL;
	ready: BOOL;
	work: BOOL;
	avar: BOOL;
	avar_vl: BOOL;
END_VAR

VAR
	prom1: BOOL;

	ftrig: F_TRIG;
	SR: SR;
END_VAR
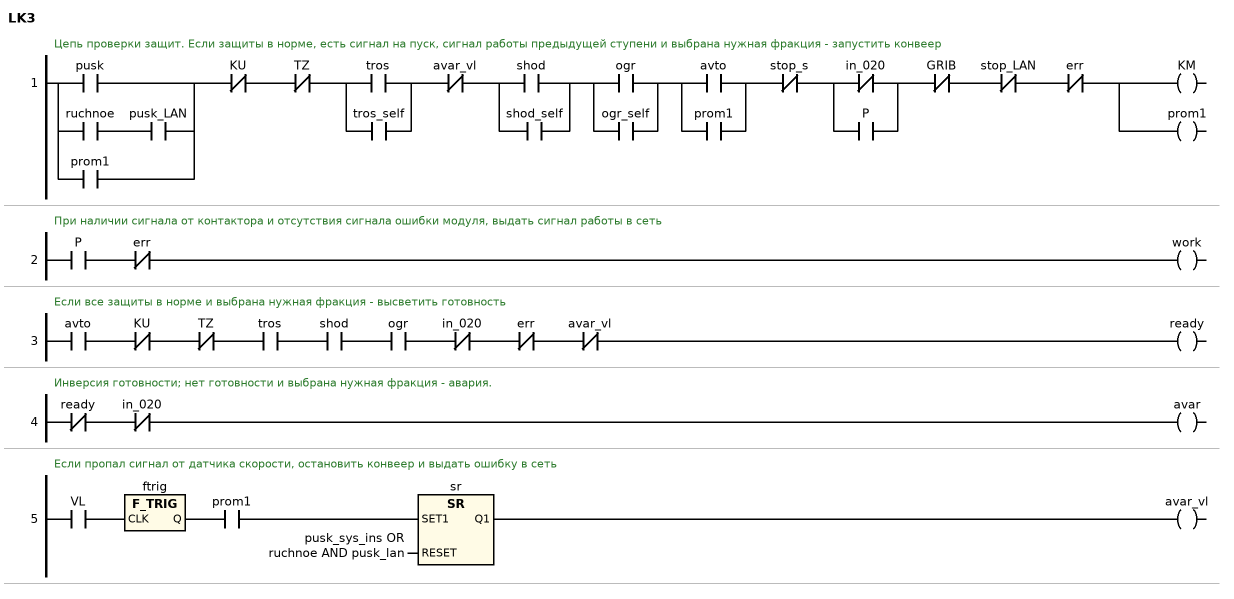
_LD_ (* Ladder Diagram *)
NETWORK 1 (* Цепь проверки защит. Если защиты в норме, есть сигнал на пуск, сигнал работы предыдущей ступени и выбрана нужная фракция - запустить конвеер *)
	{ [pusk] | [ruchnoe] - [pusk_LAN] | [prom1] } - [/KU] - [/TZ] - { [tros] | [tros_self] } - [/avar_vl] - { [shod] | [shod_self] } - { [ogr] | [ogr_self] } - { [avto] | [prom1] } - [/stop_s] - { [/in_020] | [P] } - [/GRIB] - [/stop_LAN] - [/err] --- (KM) (prom1)
NETWORK 2 (* При наличии сигнала от контактора и отсутствия сигнала ошибки модуля, выдать сигнал работы в сеть *)
	[P] - [/err] --- (work)
NETWORK 3 (* Если все защиты в норме и выбрана нужная фракция - высветить готовность *)
	[avto] - [/KU] - [/TZ] - [tros] - [shod] - [ogr] - [/in_020] - [/err] - [/avar_vl] --- (ready)
NETWORK 4 (* Инверсия готовности; нет готовности и выбрана нужная фракция - авария. *)
	[/ready] - [/in_020] --- (avar)
NETWORK 5 (* Если пропал сигнал от датчика скорости, остановить конвеер и выдать ошибку в сеть *)
	[VL] - ftrig:F_TRIG(CLK: *) - [prom1] - sr:SR(SET1: *, RESET: pusk_sys_ins OR ruchnoe AND pusk_lan) --- (avar_vl)
_END_LD_
(* the same logic as Structured Text *)
(* Network 1: Цепь проверки защит. Если защиты в норме, есть сигнал на пуск, сигнал работы предыдущей ступени и выбрана нужная фракция - запустить конвеер *)
KM := (pusk OR ruchnoe AND pusk_LAN OR prom1) AND NOT KU AND NOT TZ AND (tros OR tros_self) AND NOT avar_vl AND (shod OR shod_self) AND (ogr OR ogr_self) AND (avto OR prom1) AND NOT stop_s AND (NOT in_020 OR P) AND NOT GRIB AND NOT stop_LAN AND NOT err;
prom1 := KM;
(* Network 2: При наличии сигнала от контактора и отсутствия сигнала ошибки модуля, выдать сигнал работы в сеть *)
work := P AND NOT err;
(* Network 3: Если все защиты в норме и выбрана нужная фракция - высветить готовность *)
ready := avto AND NOT KU AND NOT TZ AND tros AND shod AND ogr AND NOT in_020 AND NOT err AND NOT avar_vl;
(* Network 4: Инверсия готовности; нет готовности и выбрана нужная фракция - авария. *)
avar := NOT ready AND NOT in_020;
(* Network 5: Если пропал сигнал от датчика скорости, остановить конвеер и выдать ошибку в сеть *)
ftrig(CLK := VL);
sr(SET1 := ftrig.Q AND prom1, RESET := pusk_sys_ins OR ruchnoe AND pusk_lan);
avar_vl := sr.Q1;
END_FUNCTION_BLOCK

(* POU counter_lk5, LD *)
FUNCTION_BLOCK counter_lk5
VAR_INPUT
	Vl: WORD;
	work: BOOL;
	in_time: WORD;
END_VAR
VAR_OUTPUT
	out_Vl: BOOL;
END_VAR
VAR
	vl_ins: WORD;
	vl_eq: BOOL;
	ton1: TOF;
	blink1: BLINK;
	tp1: TP;
	vl_sub: WORD;
	ins_time: WORD;
	time_read: TIME;
END_VAR
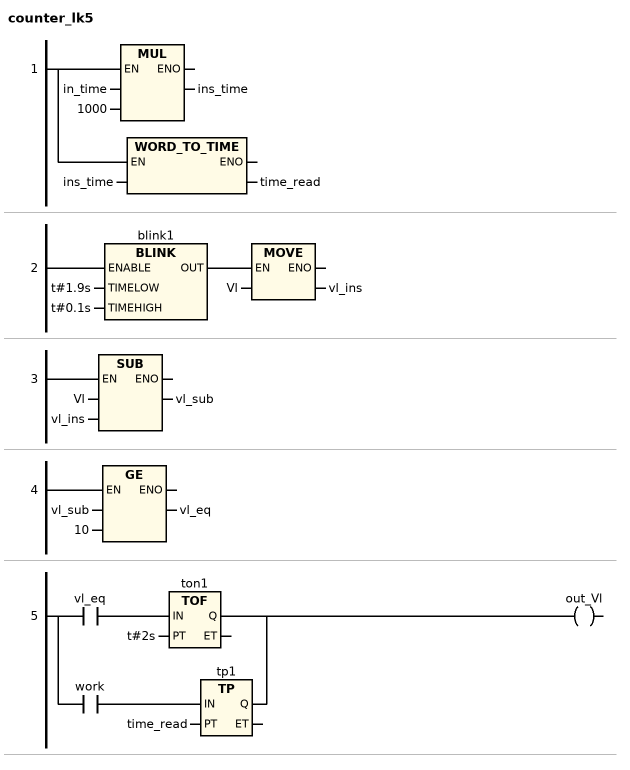
_LD_ (* Ladder Diagram *)
NETWORK 1
	*
		EN --- MUL(in_time, 1000) => ins_time
		EN --- WORD_TO_TIME(ins_time) => time_read
NETWORK 2
	blink1:BLINK(ENABLE: *, TIMELOW: t#1.9s, TIMEHIGH: t#0.1s)
		EN --- MOVE(Vl) => vl_ins
NETWORK 3
	*
		EN --- SUB(Vl, vl_ins) => vl_sub
NETWORK 4
	*
		EN --- GE(vl_sub, 10) => vl_eq
NETWORK 5
	{ [vl_eq] - ton1:TOF(IN: *, PT: t#2s) | [work] - tp1:TP(IN: *, PT: time_read) } --- (out_Vl)
_END_LD_
(* the same logic as Structured Text *)
(* Network 1 *)
ins_time := in_time * 1000;
time_read := WORD_TO_TIME(ins_time);
(* Network 2 *)
blink1(ENABLE := TRUE, TIMELOW := t#1.9s, TIMEHIGH := t#0.1s);
IF blink1.OUT THEN
	vl_ins := Vl;
END_IF;
(* Network 3 *)
vl_sub := Vl - vl_ins;
(* Network 4 *)
vl_eq := vl_sub >= 10;
(* Network 5 *)
ton1(IN := vl_eq, PT := t#2s);
tp1(IN := work, PT := time_read);
out_Vl := ton1.Q OR tp1.Q;
END_FUNCTION_BLOCK

(* POU LP1_3, LD *)
FUNCTION_BLOCK LP1_3
VAR_INPUT
	pusk_sys: BOOL;
	Vl1: BOOL;
	Vl2: BOOL;
	Vl3: BOOL;
	in_020: BOOL;
	in_040: BOOL;
	in_020_4070: BOOL;
	KU: BOOL;
	TZ1: BOOL;
	TZ2: BOOL;
	TZ3: BOOL;
	PRO: BOOL;
	avto:BOOL;
	P: BOOL;
	stop2: BOOL;
	GRIB: BOOL;
	stop_s: BOOL;
	ruchnoe: BOOL;
	pusk_LAN: BOOL;
	stop_LAN: BOOL;
	err: BOOL;
	pusk_sys_ins:BOOL;
END_VAR
VAR_OUTPUT
	KM1: BOOL;
	KM2: BOOL;
	KM4: BOOL;
	KM5: BOOL;
	KM3: BOOL;
	ready: BOOL;
	work: BOOL;
	avar: BOOL;
	avar_vl: BOOL;
END_VAR
VAR
	prom1: BOOL;
	in_020_ins: BOOL;
	in_040_ins: BOOL;
	in_020_4070_ins: BOOL;

	ftrig: F_TRIG;
	SR: SR;
END_VAR
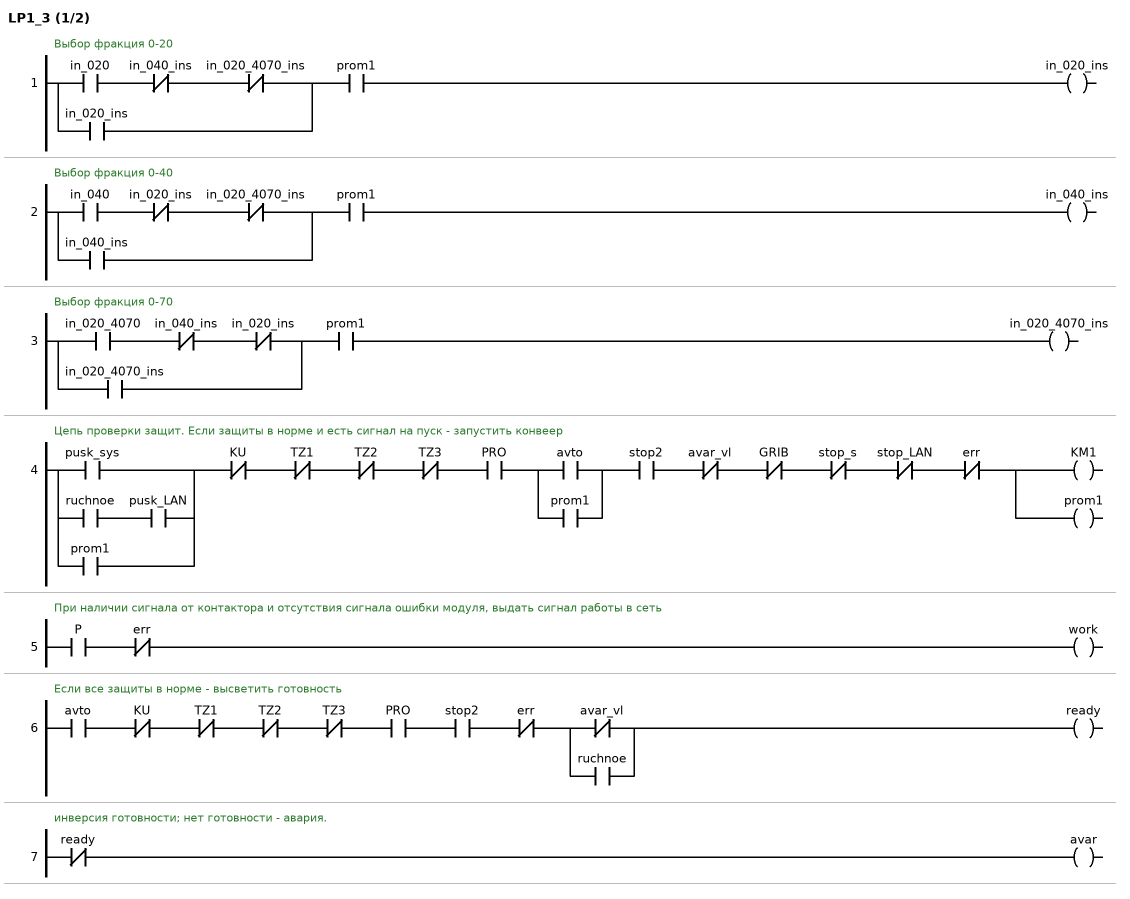
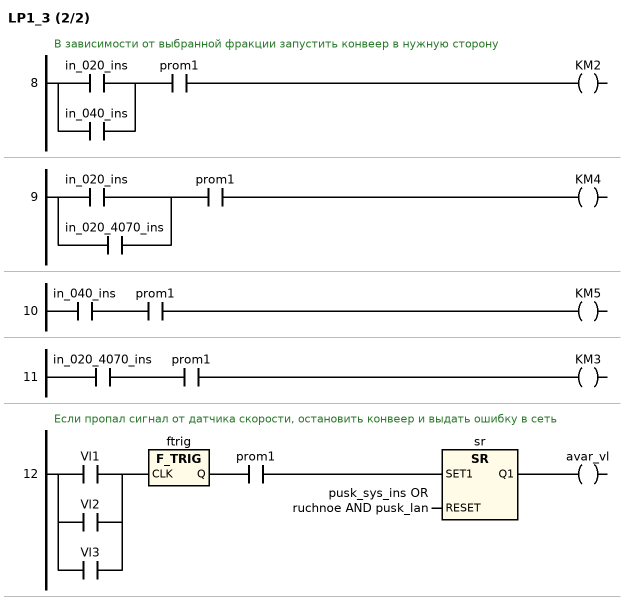
_LD_ (* Ladder Diagram *)
NETWORK 1 (* Выбор фракция 0-20 *)
	{ [in_020] - [/in_040_ins] - [/in_020_4070_ins] | [in_020_ins] } - [prom1] --- (in_020_ins)
NETWORK 2 (* Выбор фракция 0-40 *)
	{ [in_040] - [/in_020_ins] - [/in_020_4070_ins] | [in_040_ins] } - [prom1] --- (in_040_ins)
NETWORK 3 (* Выбор фракция 0-70 *)
	{ [in_020_4070] - [/in_040_ins] - [/in_020_ins] | [in_020_4070_ins] } - [prom1] --- (in_020_4070_ins)
NETWORK 4 (* Цепь проверки защит. Если защиты в норме и есть сигнал на пуск - запустить конвеер *)
	{ [pusk_sys] | [ruchnoe] - [pusk_LAN] | [prom1] } - [/KU] - [/TZ1] - [/TZ2] - [/TZ3] - [PRO] - { [avto] | [prom1] } - [stop2] - [/avar_vl] - [/GRIB] - [/stop_s] - [/stop_LAN] - [/err] --- (KM1) (prom1)
NETWORK 5 (* При наличии сигнала от контактора и отсутствия сигнала ошибки модуля, выдать сигнал работы в сеть *)
	[P] - [/err] --- (work)
NETWORK 6 (* Если все защиты в норме - высветить готовность *)
	[avto] - [/KU] - [/TZ1] - [/TZ2] - [/TZ3] - [PRO] - [stop2] - [/err] - { [/avar_vl] | [ruchnoe] } --- (ready)
NETWORK 7 (* инверсия готовности; нет готовности - авария. *)
	[/ready] --- (avar)
NETWORK 8 (* В зависимости от выбранной фракции запустить конвеер в нужную сторону *)
	{ [in_020_ins] | [in_040_ins] } - [prom1] --- (KM2)
NETWORK 9
	{ [in_020_ins] | [in_020_4070_ins] } - [prom1] --- (KM4)
NETWORK 10
	[in_040_ins] - [prom1] --- (KM5)
NETWORK 11
	[in_020_4070_ins] - [prom1] --- (KM3)
NETWORK 12 (* Если пропал сигнал от датчика скорости, остановить конвеер и выдать ошибку в сеть *)
	{ [Vl1] | [Vl2] | [Vl3] } - ftrig:F_TRIG(CLK: *) - [prom1] - sr:SR(SET1: *, RESET: pusk_sys_ins OR ruchnoe AND pusk_lan) --- (avar_vl)
_END_LD_
(* the same logic as Structured Text *)
(* Network 1: Выбор фракция 0-20 *)
in_020_ins := (in_020 AND NOT in_040_ins AND NOT in_020_4070_ins OR in_020_ins) AND prom1;
(* Network 2: Выбор фракция 0-40 *)
in_040_ins := (in_040 AND NOT in_020_ins AND NOT in_020_4070_ins OR in_040_ins) AND prom1;
(* Network 3: Выбор фракция 0-70 *)
in_020_4070_ins := (in_020_4070 AND NOT in_040_ins AND NOT in_020_ins OR in_020_4070_ins) AND prom1;
(* Network 4: Цепь проверки защит. Если защиты в норме и есть сигнал на пуск - запустить конвеер *)
KM1 := (pusk_sys OR ruchnoe AND pusk_LAN OR prom1) AND NOT KU AND NOT TZ1 AND NOT TZ2 AND NOT TZ3 AND PRO AND (avto OR prom1) AND stop2 AND NOT avar_vl AND NOT GRIB AND NOT stop_s AND NOT stop_LAN AND NOT err;
prom1 := KM1;
(* Network 5: При наличии сигнала от контактора и отсутствия сигнала ошибки модуля, выдать сигнал работы в сеть *)
work := P AND NOT err;
(* Network 6: Если все защиты в норме - высветить готовность *)
ready := avto AND NOT KU AND NOT TZ1 AND NOT TZ2 AND NOT TZ3 AND PRO AND stop2 AND NOT err AND (NOT avar_vl OR ruchnoe);
(* Network 7: инверсия готовности; нет готовности - авария. *)
avar := NOT ready;
(* Network 8: В зависимости от выбранной фракции запустить конвеер в нужную сторону *)
KM2 := (in_020_ins OR in_040_ins) AND prom1;
(* Network 9 *)
KM4 := (in_020_ins OR in_020_4070_ins) AND prom1;
(* Network 10 *)
KM5 := in_040_ins AND prom1;
(* Network 11 *)
KM3 := in_020_4070_ins AND prom1;
(* Network 12: Если пропал сигнал от датчика скорости, остановить конвеер и выдать ошибку в сеть *)
ftrig(CLK := Vl1 OR Vl2 OR Vl3);
sr(SET1 := ftrig.Q AND prom1, RESET := pusk_sys_ins OR ruchnoe AND pusk_lan);
avar_vl := sr.Q1;
END_FUNCTION_BLOCK

(* POU Grohot1, LD *)
FUNCTION_BLOCK Grohot1
VAR_INPUT
	pusk: BOOL;
	avto: BOOL;
	KU: BOOL;
	TZ: BOOL;
	P:BOOL;
	STOP: BOOL;
	stop_sys: BOOL;
	GRIB: BOOL;
	stop_lv: BOOL;
	ruchnoe: BOOL;
	pusk_LAN: BOOL;
	stop_LAN: BOOL;
	err: BOOL;
END_VAR

VAR_OUTPUT
	KM: BOOL;
	ready: BOOL;
	work: BOOL;
	avar: BOOL;
END_VAR

VAR
	prom1: BOOL;
END_VAR
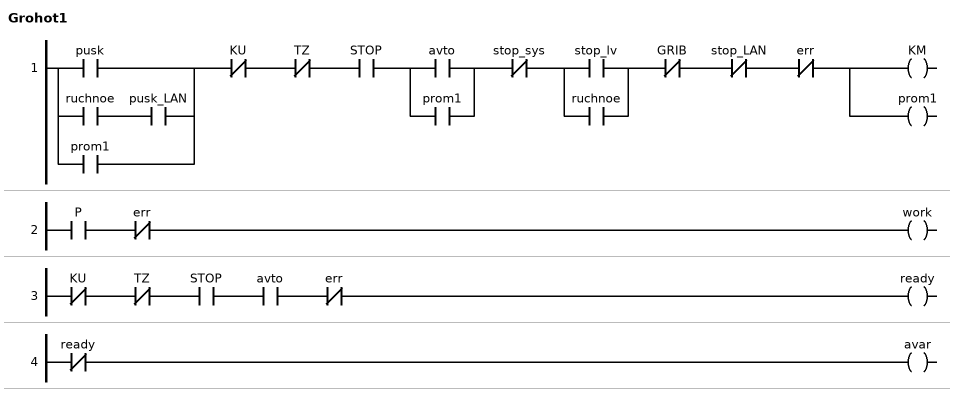
_LD_ (* Ladder Diagram *)
NETWORK 1
	{ [pusk] | [ruchnoe] - [pusk_LAN] | [prom1] } - [/KU] - [/TZ] - [STOP] - { [avto] | [prom1] } - [/stop_sys] - { [stop_lv] | [ruchnoe] } - [/GRIB] - [/stop_LAN] - [/err] --- (KM) (prom1)
NETWORK 2
	[P] - [/err] --- (work)
NETWORK 3
	[/KU] - [/TZ] - [STOP] - [avto] - [/err] --- (ready)
NETWORK 4
	[/ready] --- (avar)
_END_LD_
(* the same logic as Structured Text *)
(* Network 1 *)
KM := (pusk OR ruchnoe AND pusk_LAN OR prom1) AND NOT KU AND NOT TZ AND STOP AND (avto OR prom1) AND NOT stop_sys AND (stop_lv OR ruchnoe) AND NOT GRIB AND NOT stop_LAN AND NOT err;
prom1 := KM;
(* Network 2 *)
work := P AND NOT err;
(* Network 3 *)
ready := NOT KU AND NOT TZ AND STOP AND avto AND NOT err;
(* Network 4 *)
avar := NOT ready;
END_FUNCTION_BLOCK

(* POU LP4, LD *)
FUNCTION_BLOCK LP4
VAR_INPUT
	pusk: BOOL;
	avto: BOOL;
	STOP: BOOL;
	VL: BOOL;
	MD2: BOOL;
	stop_lv:BOOL;
	GRIB: BOOL;
	input_Hz: WORD;
	stop_s: BOOL;
	pusk_LAN: BOOL;
	stop_LAN: BOOL;
	P: WORD;
	ruchnoe: BOOL;
	err: BOOL;
	pusk_sys_ins: BOOL;
	avar_FC: BOOL;
	err_temp: BOOL;
END_VAR

VAR_OUTPUT
	ready: BOOL;
	KM: WORD;
	work: BOOL;
	avar: BOOL;
	met: BOOL;
	b1_00: WORD;
	b1_04: WORD;
	avto_in: BOOL;
	avar_vl: BOOL;
END_VAR

VAR
	prom1: BOOL;
	Hz: WORD;
	ftrig: F_TRIG;
	SR: SR;
END_VAR
VAR (* helpers for the ST form of the networks *)
	_p1 : BOOL;
END_VAR
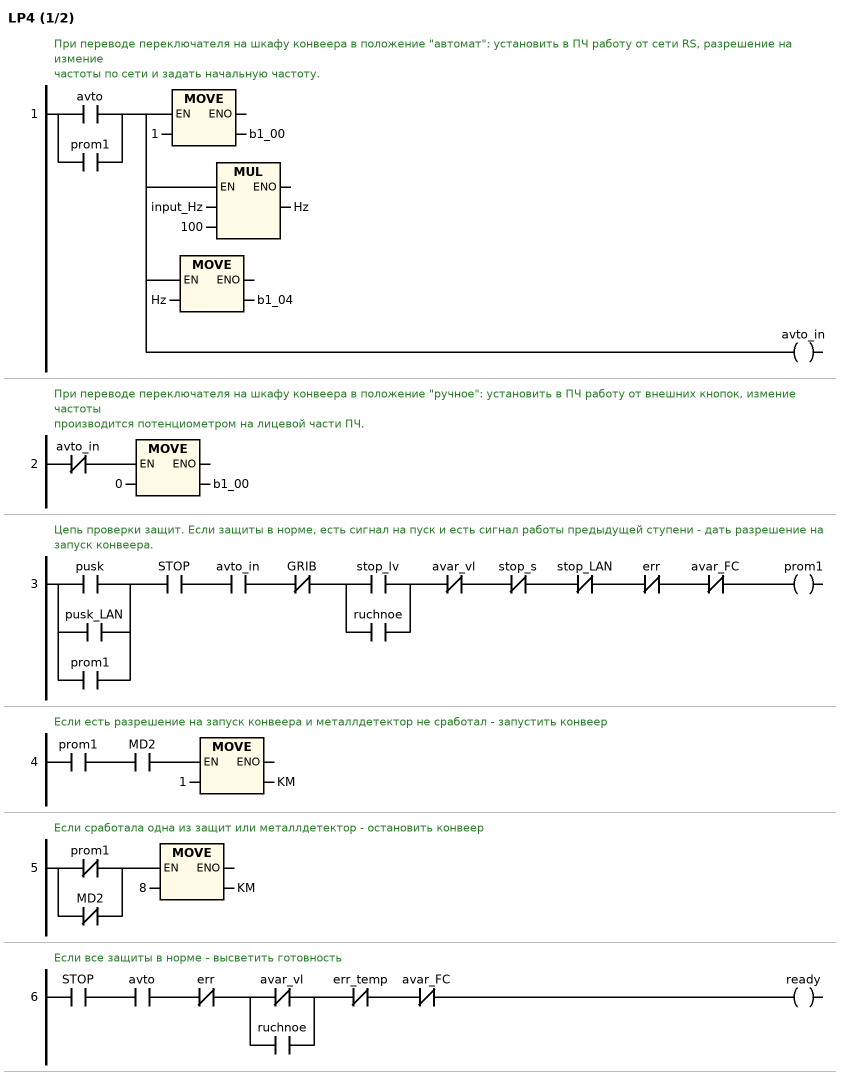
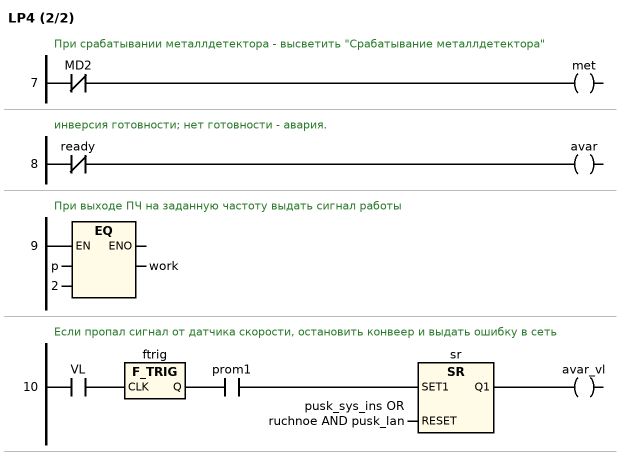
_LD_ (* Ladder Diagram *)
NETWORK 1 (* При переводе переключателя на шкафу конвеера в положение "автомат": установить в ПЧ работу от сети RS, разрешение на измение / частоты по сети и задать начальную частоту. *)
	{ [avto] | [prom1] } --- (avto_in)
		EN --- MOVE(1) => b1_00
		EN --- MUL(input_Hz, 100) => Hz
		EN --- MOVE(Hz) => b1_04
NETWORK 2 (* При переводе переключателя на шкафу конвеера в положение "ручное": установить в ПЧ работу от внешних кнопок, измение частоты / производится потенциометром на лицевой части ПЧ. *)
	[/avto_in]
		EN --- MOVE(0) => b1_00
NETWORK 3 (* Цепь проверки защит. Если защиты в норме, есть сигнал на пуск и есть сигнал работы предыдущей ступени - дать разрешение на запуск конвеера. *)
	{ [pusk] | [pusk_LAN] | [prom1] } - [STOP] - [avto_in] - [/GRIB] - { [stop_lv] | [ruchnoe] } - [/avar_vl] - [/stop_s] - [/stop_LAN] - [/err] - [/avar_FC] --- (prom1)
NETWORK 4 (* Если есть разрешение на запуск конвеера и металлдетектор не сработал - запустить конвеер *)
	[prom1] - [MD2]
		EN --- MOVE(1) => KM
NETWORK 5 (* Если сработала одна из защит или металлдетектор - остановить конвеер *)
	{ [/prom1] | [/MD2] }
		EN --- MOVE(8) => KM
NETWORK 6 (* Если все защиты в норме - высветить готовность *)
	[STOP] - [avto] - [/err] - { [/avar_vl] | [ruchnoe] } - [/err_temp] - [/avar_FC] --- (ready)
NETWORK 7 (* При срабатывании металлдетектора - высветить "Срабатывание металлдетектора" *)
	[/MD2] --- (met)
NETWORK 8 (* инверсия готовности; нет готовности - авария. *)
	[/ready] --- (avar)
NETWORK 9 (* При выходе ПЧ на заданную частоту выдать сигнал работы *)
	*
		EN --- EQ(p, 2) => work
NETWORK 10 (* Если пропал сигнал от датчика скорости, остановить конвеер и выдать ошибку в сеть *)
	[VL] - ftrig:F_TRIG(CLK: *) - [prom1] - sr:SR(SET1: *, RESET: pusk_sys_ins OR ruchnoe AND pusk_lan) --- (avar_vl)
_END_LD_
(* the same logic as Structured Text *)
(* Network 1: При переводе переключателя на шкафу конвеера в положение "автомат": установить в ПЧ работу от сети RS, разрешение на измение / частоты по сети и задать начальную частоту. *)
_p1 := avto OR prom1;
IF _p1 THEN
	b1_00 := 1;
	Hz := input_Hz * 100;
	b1_04 := Hz;
END_IF;
avto_in := _p1;
(* Network 2: При переводе переключателя на шкафу конвеера в положение "ручное": установить в ПЧ работу от внешних кнопок, измение частоты / производится потенциометром на лицевой части ПЧ. *)
IF NOT avto_in THEN
	b1_00 := 0;
END_IF;
(* Network 3: Цепь проверки защит. Если защиты в норме, есть сигнал на пуск и есть сигнал работы предыдущей ступени - дать разрешение на запуск конвеера. *)
prom1 := (pusk OR pusk_LAN OR prom1) AND STOP AND avto_in AND NOT GRIB AND (stop_lv OR ruchnoe) AND NOT avar_vl AND NOT stop_s AND NOT stop_LAN AND NOT err AND NOT avar_FC;
(* Network 4: Если есть разрешение на запуск конвеера и металлдетектор не сработал - запустить конвеер *)
IF prom1 AND MD2 THEN
	KM := 1;
END_IF;
(* Network 5: Если сработала одна из защит или металлдетектор - остановить конвеер *)
IF NOT prom1 OR NOT MD2 THEN
	KM := 8;
END_IF;
(* Network 6: Если все защиты в норме - высветить готовность *)
ready := STOP AND avto AND NOT err AND (NOT avar_vl OR ruchnoe) AND NOT err_temp AND NOT avar_FC;
(* Network 7: При срабатывании металлдетектора - высветить "Срабатывание металлдетектора" *)
met := NOT MD2;
(* Network 8: инверсия готовности; нет готовности - авария. *)
avar := NOT ready;
(* Network 9: При выходе ПЧ на заданную частоту выдать сигнал работы *)
work := p = 2;
(* Network 10: Если пропал сигнал от датчика скорости, остановить конвеер и выдать ошибку в сеть *)
ftrig(CLK := VL);
sr(SET1 := ftrig.Q AND prom1, RESET := pusk_sys_ins OR ruchnoe AND pusk_lan);
avar_vl := sr.Q1;
END_FUNCTION_BLOCK

(* POU LP4_without_FC, LD *)
FUNCTION_BLOCK LP4_without_FC (*функциональный блок управления ленточным конвеером 4 с металлодетектором*)
VAR_INPUT
	pusk: BOOL;
	avto:BOOL;
	KU: BOOL;
	TZ: BOOL;
	MD3: BOOL;
	P: BOOL;
	stop_lv: BOOL;
	GRIB: BOOL;
	stop_s: BOOL;
	ruchnoe: BOOL;
	pusk_LAN: BOOL;
	stop_LAN: BOOL;
	err: BOOL;
END_VAR

VAR_OUTPUT
	KM:BOOL;
	ready: BOOL;
	work: BOOL;
	avar: BOOL;
	metall_LK4: BOOL;
END_VAR

VAR
	prom1: BOOL;
END_VAR
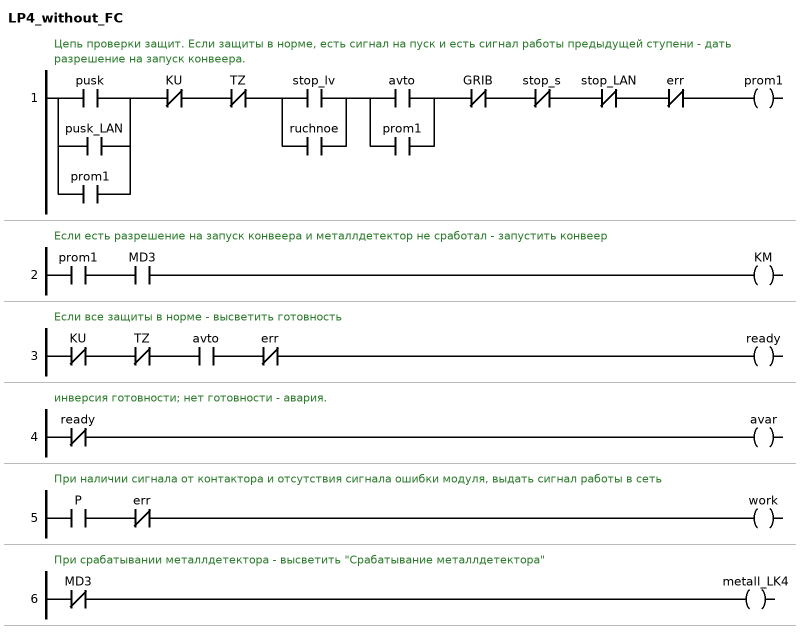
_LD_ (* Ladder Diagram *)
NETWORK 1 (* Цепь проверки защит. Если защиты в норме, есть сигнал на пуск и есть сигнал работы предыдущей ступени - дать разрешение на запуск конвеера. *)
	{ [pusk] | [pusk_LAN] | [prom1] } - [/KU] - [/TZ] - { [stop_lv] | [ruchnoe] } - { [avto] | [prom1] } - [/GRIB] - [/stop_s] - [/stop_LAN] - [/err] --- (prom1)
NETWORK 2 (* Если есть разрешение на запуск конвеера и металлдетектор не сработал - запустить конвеер *)
	[prom1] - [MD3] --- (KM)
NETWORK 3 (* Если все защиты в норме - высветить готовность *)
	[/KU] - [/TZ] - [avto] - [/err] --- (ready)
NETWORK 4 (* инверсия готовности; нет готовности - авария. *)
	[/ready] --- (avar)
NETWORK 5 (* При наличии сигнала от контактора и отсутствия сигнала ошибки модуля, выдать сигнал работы в сеть *)
	[P] - [/err] --- (work)
NETWORK 6 (* При срабатывании металлдетектора - высветить "Срабатывание металлдетектора" *)
	[/MD3] --- (metall_LK4)
_END_LD_
(* the same logic as Structured Text *)
(* Network 1: Цепь проверки защит. Если защиты в норме, есть сигнал на пуск и есть сигнал работы предыдущей ступени - дать разрешение на запуск конвеера. *)
prom1 := (pusk OR pusk_LAN OR prom1) AND NOT KU AND NOT TZ AND (stop_lv OR ruchnoe) AND (avto OR prom1) AND NOT GRIB AND NOT stop_s AND NOT stop_LAN AND NOT err;
(* Network 2: Если есть разрешение на запуск конвеера и металлдетектор не сработал - запустить конвеер *)
KM := prom1 AND MD3;
(* Network 3: Если все защиты в норме - высветить готовность *)
ready := NOT KU AND NOT TZ AND avto AND NOT err;
(* Network 4: инверсия готовности; нет готовности - авария. *)
avar := NOT ready;
(* Network 5: При наличии сигнала от контактора и отсутствия сигнала ошибки модуля, выдать сигнал работы в сеть *)
work := P AND NOT err;
(* Network 6: При срабатывании металлдетектора - высветить "Срабатывание металлдетектора" *)
metall_LK4 := NOT MD3;
END_FUNCTION_BLOCK

(* POU LP5, LD *)
FUNCTION_BLOCK LP5
VAR_INPUT
	pusk: BOOL;
	avto: BOOL;
	STOP: BOOL;
	VL: BOOL;
	MD2: BOOL;
	stop_lv:BOOL;
	GRIB: BOOL;
	input_Hz: WORD;
	stop_s: BOOL;
	pusk_LAN: BOOL;
	stop_LAN: BOOL;
	P: WORD;
	ruchnoe: BOOL;
	ins_0_40: BOOL;
	err: BOOL;
	pusk_sys_ins: BOOL;
	avar_FC: BOOL;
END_VAR

VAR_OUTPUT
	ready: BOOL;
	KM: WORD;
	work: BOOL;
	avar: BOOL;
	met: BOOL;
	b1_00: WORD;
	b1_04: WORD;
	avto_in: BOOL;
	avar_vl: BOOL;
END_VAR

VAR
	prom1: BOOL;
	Hz: WORD;
	ftrig: F_TRIG;
	SR: SR;
END_VAR
VAR (* helpers for the ST form of the networks *)
	_p1 : BOOL;
END_VAR
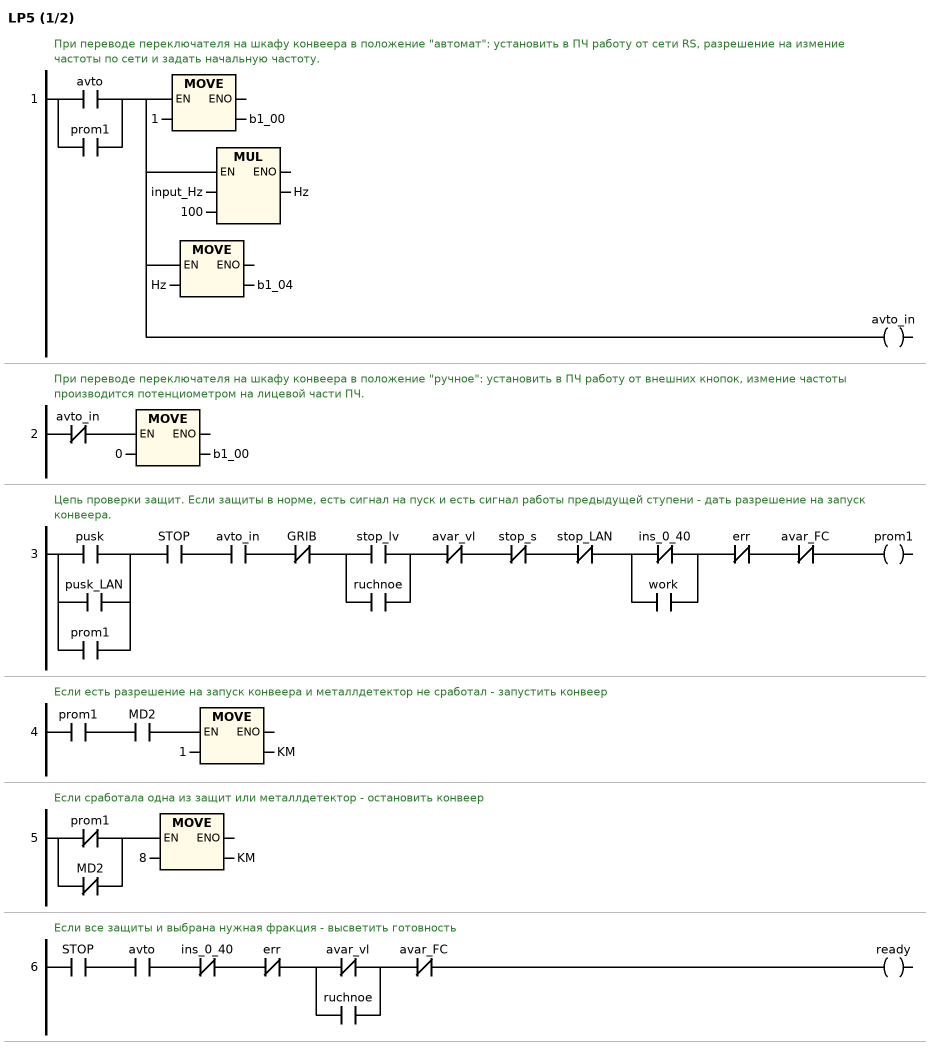
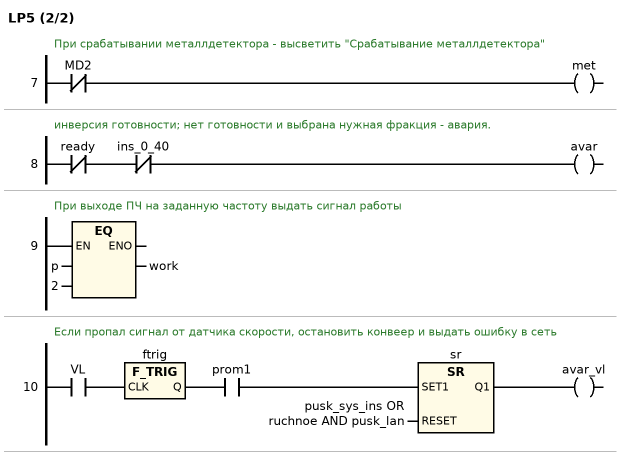
_LD_ (* Ladder Diagram *)
NETWORK 1 (* При переводе переключателя на шкафу конвеера в положение "автомат": установить в ПЧ работу от сети RS, разрешение на измение / частоты по сети и задать начальную частоту. *)
	{ [avto] | [prom1] } --- (avto_in)
		EN --- MOVE(1) => b1_00
		EN --- MUL(input_Hz, 100) => Hz
		EN --- MOVE(Hz) => b1_04
NETWORK 2 (* При переводе переключателя на шкафу конвеера в положение "ручное": установить в ПЧ работу от внешних кнопок, измение частоты / производится потенциометром на лицевой части ПЧ. *)
	[/avto_in]
		EN --- MOVE(0) => b1_00
NETWORK 3 (* Цепь проверки защит. Если защиты в норме, есть сигнал на пуск и есть сигнал работы предыдущей ступени - дать разрешение на запуск конвеера. *)
	{ [pusk] | [pusk_LAN] | [prom1] } - [STOP] - [avto_in] - [/GRIB] - { [stop_lv] | [ruchnoe] } - [/avar_vl] - [/stop_s] - [/stop_LAN] - { [/ins_0_40] | [work] } - [/err] - [/avar_FC] --- (prom1)
NETWORK 4 (* Если есть разрешение на запуск конвеера и металлдетектор не сработал - запустить конвеер *)
	[prom1] - [MD2]
		EN --- MOVE(1) => KM
NETWORK 5 (* Если сработала одна из защит или металлдетектор - остановить конвеер *)
	{ [/prom1] | [/MD2] }
		EN --- MOVE(8) => KM
NETWORK 6 (* Если все защиты и выбрана нужная фракция - высветить готовность *)
	[STOP] - [avto] - [/ins_0_40] - [/err] - { [/avar_vl] | [ruchnoe] } - [/avar_FC] --- (ready)
NETWORK 7 (* При срабатывании металлдетектора - высветить "Срабатывание металлдетектора" *)
	[/MD2] --- (met)
NETWORK 8 (* инверсия готовности; нет готовности и выбрана нужная фракция - авария. *)
	[/ready] - [/ins_0_40] --- (avar)
NETWORK 9 (* При выходе ПЧ на заданную частоту выдать сигнал работы *)
	*
		EN --- EQ(p, 2) => work
NETWORK 10 (* Если пропал сигнал от датчика скорости, остановить конвеер и выдать ошибку в сеть *)
	[VL] - ftrig:F_TRIG(CLK: *) - [prom1] - sr:SR(SET1: *, RESET: pusk_sys_ins OR ruchnoe AND pusk_lan) --- (avar_vl)
_END_LD_
(* the same logic as Structured Text *)
(* Network 1: При переводе переключателя на шкафу конвеера в положение "автомат": установить в ПЧ работу от сети RS, разрешение на измение / частоты по сети и задать начальную частоту. *)
_p1 := avto OR prom1;
IF _p1 THEN
	b1_00 := 1;
	Hz := input_Hz * 100;
	b1_04 := Hz;
END_IF;
avto_in := _p1;
(* Network 2: При переводе переключателя на шкафу конвеера в положение "ручное": установить в ПЧ работу от внешних кнопок, измение частоты / производится потенциометром на лицевой части ПЧ. *)
IF NOT avto_in THEN
	b1_00 := 0;
END_IF;
(* Network 3: Цепь проверки защит. Если защиты в норме, есть сигнал на пуск и есть сигнал работы предыдущей ступени - дать разрешение на запуск конвеера. *)
prom1 := (pusk OR pusk_LAN OR prom1) AND STOP AND avto_in AND NOT GRIB AND (stop_lv OR ruchnoe) AND NOT avar_vl AND NOT stop_s AND NOT stop_LAN AND (NOT ins_0_40 OR work) AND NOT err AND NOT avar_FC;
(* Network 4: Если есть разрешение на запуск конвеера и металлдетектор не сработал - запустить конвеер *)
IF prom1 AND MD2 THEN
	KM := 1;
END_IF;
(* Network 5: Если сработала одна из защит или металлдетектор - остановить конвеер *)
IF NOT prom1 OR NOT MD2 THEN
	KM := 8;
END_IF;
(* Network 6: Если все защиты и выбрана нужная фракция - высветить готовность *)
ready := STOP AND avto AND NOT ins_0_40 AND NOT err AND (NOT avar_vl OR ruchnoe) AND NOT avar_FC;
(* Network 7: При срабатывании металлдетектора - высветить "Срабатывание металлдетектора" *)
met := NOT MD2;
(* Network 8: инверсия готовности; нет готовности и выбрана нужная фракция - авария. *)
avar := NOT ready AND NOT ins_0_40;
(* Network 9: При выходе ПЧ на заданную частоту выдать сигнал работы *)
work := p = 2;
(* Network 10: Если пропал сигнал от датчика скорости, остановить конвеер и выдать ошибку в сеть *)
ftrig(CLK := VL);
sr(SET1 := ftrig.Q AND prom1, RESET := pusk_sys_ins OR ruchnoe AND pusk_lan);
avar_vl := sr.Q1;
END_FUNCTION_BLOCK

(* POU LK4, LD *)
FUNCTION_BLOCK LK4 (*функциональный блок управления ленточным конвеером 4 с металлодетектором*)
VAR_INPUT
	pusk: BOOL;
	avto:BOOL;
	KU: BOOL;
	TZ: BOOL;
	tros: BOOL;
	shod: BOOL;
	MD3: BOOL;
	VL:BOOL;
	P: BOOL;
	stop_lv: BOOL;
	GRIB: BOOL;
	stop_s: BOOL;
	ruchnoe: BOOL;
	pusk_LAN: BOOL;
	stop_LAN: BOOL;
	err: BOOL;
	tros_self: BOOL;
	shod_self: BOOL;
	pusk_sys_ins:BOOL;
END_VAR

VAR_OUTPUT
	KM:BOOL;
	ready: BOOL;
	work: BOOL;
	avar: BOOL;
	metall_LK4: BOOL;
	avar_vl: BOOL;
END_VAR

VAR
	prom1: BOOL;

	ftrig: F_TRIG;
	SR: SR;
END_VAR
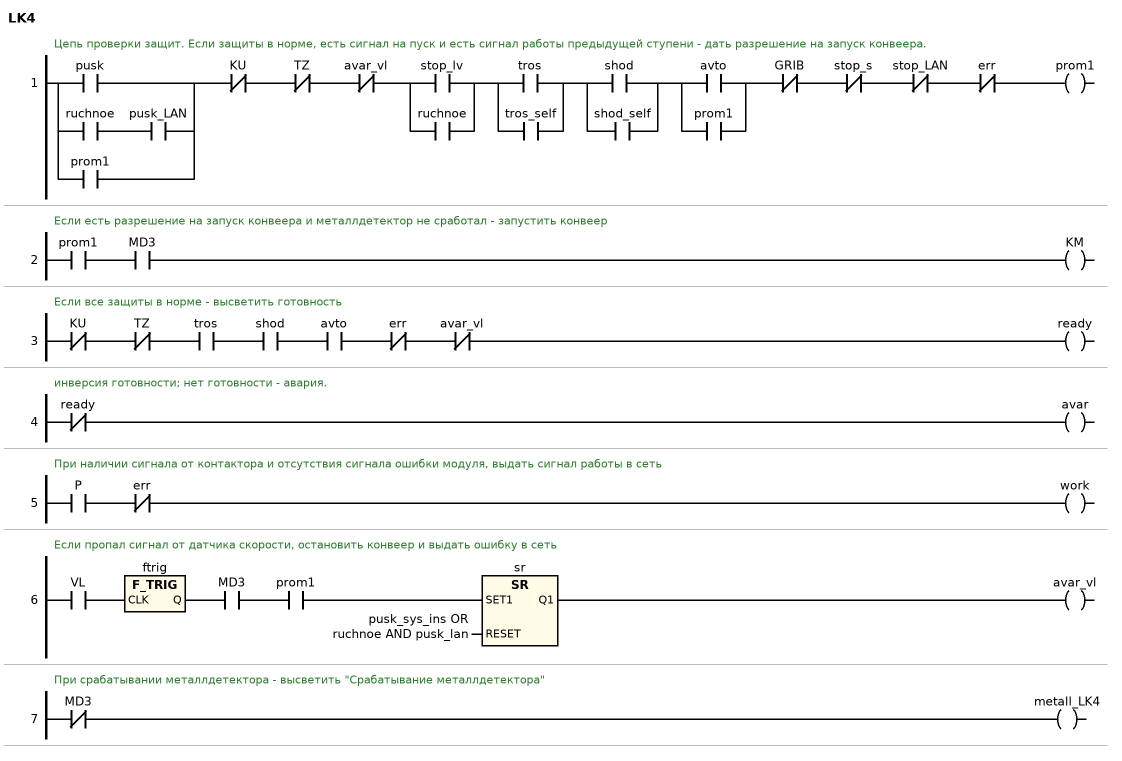
_LD_ (* Ladder Diagram *)
NETWORK 1 (* Цепь проверки защит. Если защиты в норме, есть сигнал на пуск и есть сигнал работы предыдущей ступени - дать разрешение на запуск конвеера. *)
	{ [pusk] | [ruchnoe] - [pusk_LAN] | [prom1] } - [/KU] - [/TZ] - [/avar_vl] - { [stop_lv] | [ruchnoe] } - { [tros] | [tros_self] } - { [shod] | [shod_self] } - { [avto] | [prom1] } - [/GRIB] - [/stop_s] - [/stop_LAN] - [/err] --- (prom1)
NETWORK 2 (* Если есть разрешение на запуск конвеера и металлдетектор не сработал - запустить конвеер *)
	[prom1] - [MD3] --- (KM)
NETWORK 3 (* Если все защиты в норме - высветить готовность *)
	[/KU] - [/TZ] - [tros] - [shod] - [avto] - [/err] - [/avar_vl] --- (ready)
NETWORK 4 (* инверсия готовности; нет готовности - авария. *)
	[/ready] --- (avar)
NETWORK 5 (* При наличии сигнала от контактора и отсутствия сигнала ошибки модуля, выдать сигнал работы в сеть *)
	[P] - [/err] --- (work)
NETWORK 6 (* Если пропал сигнал от датчика скорости, остановить конвеер и выдать ошибку в сеть *)
	[VL] - ftrig:F_TRIG(CLK: *) - [MD3] - [prom1] - sr:SR(SET1: *, RESET: pusk_sys_ins OR ruchnoe AND pusk_lan) --- (avar_vl)
NETWORK 7 (* При срабатывании металлдетектора - высветить "Срабатывание металлдетектора" *)
	[/MD3] --- (metall_LK4)
_END_LD_
(* the same logic as Structured Text *)
(* Network 1: Цепь проверки защит. Если защиты в норме, есть сигнал на пуск и есть сигнал работы предыдущей ступени - дать разрешение на запуск конвеера. *)
prom1 := (pusk OR ruchnoe AND pusk_LAN OR prom1) AND NOT KU AND NOT TZ AND NOT avar_vl AND (stop_lv OR ruchnoe) AND (tros OR tros_self) AND (shod OR shod_self) AND (avto OR prom1) AND NOT GRIB AND NOT stop_s AND NOT stop_LAN AND NOT err;
(* Network 2: Если есть разрешение на запуск конвеера и металлдетектор не сработал - запустить конвеер *)
KM := prom1 AND MD3;
(* Network 3: Если все защиты в норме - высветить готовность *)
ready := NOT KU AND NOT TZ AND tros AND shod AND avto AND NOT err AND NOT avar_vl;
(* Network 4: инверсия готовности; нет готовности - авария. *)
avar := NOT ready;
(* Network 5: При наличии сигнала от контактора и отсутствия сигнала ошибки модуля, выдать сигнал работы в сеть *)
work := P AND NOT err;
(* Network 6: Если пропал сигнал от датчика скорости, остановить конвеер и выдать ошибку в сеть *)
ftrig(CLK := VL);
sr(SET1 := ftrig.Q AND MD3 AND prom1, RESET := pusk_sys_ins OR ruchnoe AND pusk_lan);
avar_vl := sr.Q1;
(* Network 7: При срабатывании металлдетектора - высветить "Срабатывание металлдетектора" *)
metall_LK4 := NOT MD3;
END_FUNCTION_BLOCK

(* POU LK2, LD *)
FUNCTION_BLOCK LK2 (*Ленточные конвееры 2,5 и 9*)
VAR_INPUT
	pusk: BOOL;
	avto:BOOL;
	KU: BOOL;
	TZ: BOOL;
	tros: BOOL;
	shod: BOOL;
	ogr: BOOL;
	VL:BOOL;
	P: BOOL;
	GRIB: BOOL;
	stop_s: BOOL;
	stop_lv: BOOL;
	ruchnoe: BOOL;
	pusk_LAN: BOOL;
	stop_LAN: BOOL;
	err: BOOL;
	tros_self: BOOL;
	shod_self: BOOL;
	ogr_self: BOOL;
	pusk_sys_ins:BOOL;
END_VAR

VAR_OUTPUT
	KM:BOOL;
	ready: BOOL;
	work: BOOL;
	avar: BOOL;
	avar_vl: BOOL;
END_VAR

VAR
	prom1: BOOL;

	ftrig: F_TRIG;
	SR: SR;
END_VAR
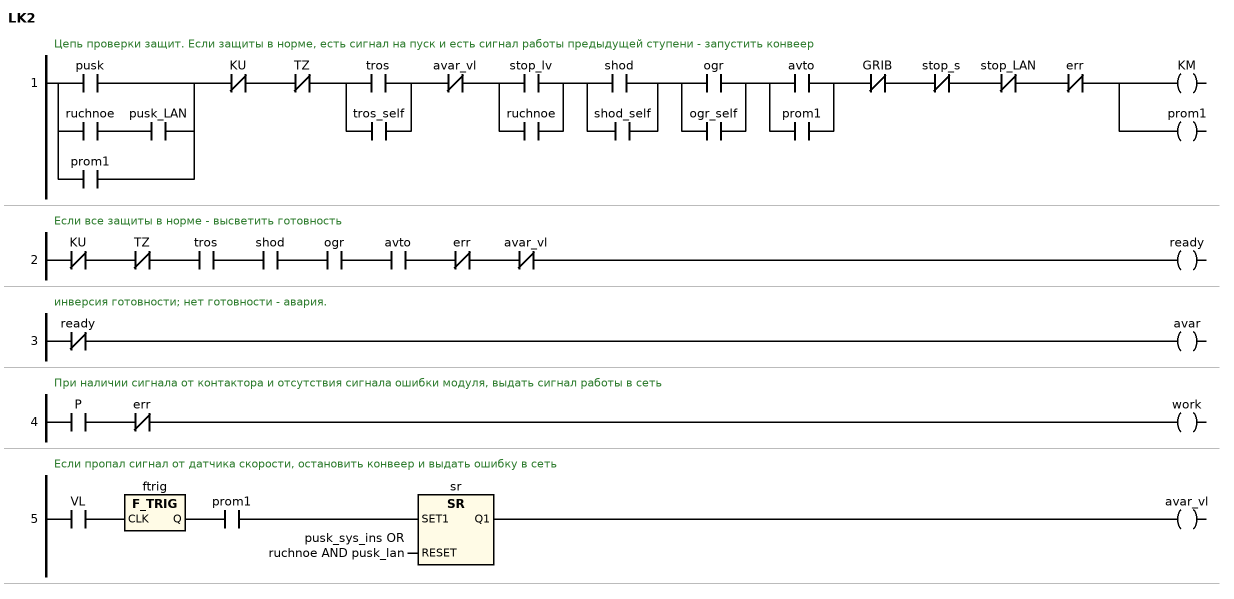
_LD_ (* Ladder Diagram *)
NETWORK 1 (* Цепь проверки защит. Если защиты в норме, есть сигнал на пуск и есть сигнал работы предыдущей ступени - запустить конвеер *)
	{ [pusk] | [ruchnoe] - [pusk_LAN] | [prom1] } - [/KU] - [/TZ] - { [tros] | [tros_self] } - [/avar_vl] - { [stop_lv] | [ruchnoe] } - { [shod] | [shod_self] } - { [ogr] | [ogr_self] } - { [avto] | [prom1] } - [/GRIB] - [/stop_s] - [/stop_LAN] - [/err] --- (KM) (prom1)
NETWORK 2 (* Если все защиты в норме - высветить готовность *)
	[/KU] - [/TZ] - [tros] - [shod] - [ogr] - [avto] - [/err] - [/avar_vl] --- (ready)
NETWORK 3 (* инверсия готовности; нет готовности - авария. *)
	[/ready] --- (avar)
NETWORK 4 (* При наличии сигнала от контактора и отсутствия сигнала ошибки модуля, выдать сигнал работы в сеть *)
	[P] - [/err] --- (work)
NETWORK 5 (* Если пропал сигнал от датчика скорости, остановить конвеер и выдать ошибку в сеть *)
	[VL] - ftrig:F_TRIG(CLK: *) - [prom1] - sr:SR(SET1: *, RESET: pusk_sys_ins OR ruchnoe AND pusk_lan) --- (avar_vl)
_END_LD_
(* the same logic as Structured Text *)
(* Network 1: Цепь проверки защит. Если защиты в норме, есть сигнал на пуск и есть сигнал работы предыдущей ступени - запустить конвеер *)
KM := (pusk OR ruchnoe AND pusk_LAN OR prom1) AND NOT KU AND NOT TZ AND (tros OR tros_self) AND NOT avar_vl AND (stop_lv OR ruchnoe) AND (shod OR shod_self) AND (ogr OR ogr_self) AND (avto OR prom1) AND NOT GRIB AND NOT stop_s AND NOT stop_LAN AND NOT err;
prom1 := KM;
(* Network 2: Если все защиты в норме - высветить готовность *)
ready := NOT KU AND NOT TZ AND tros AND shod AND ogr AND avto AND NOT err AND NOT avar_vl;
(* Network 3: инверсия готовности; нет готовности - авария. *)
avar := NOT ready;
(* Network 4: При наличии сигнала от контактора и отсутствия сигнала ошибки модуля, выдать сигнал работы в сеть *)
work := P AND NOT err;
(* Network 5: Если пропал сигнал от датчика скорости, остановить конвеер и выдать ошибку в сеть *)
ftrig(CLK := VL);
sr(SET1 := ftrig.Q AND prom1, RESET := pusk_sys_ins OR ruchnoe AND pusk_lan);
avar_vl := sr.Q1;
END_FUNCTION_BLOCK

(* POU VP1, LD *)
FUNCTION_BLOCK VP1
VAR_INPUT
	pusk: BOOL;
	avto: BOOL;
	KU: BOOL;
	TZ: BOOL;
	STOP: BOOL;
	stop_lv:BOOL;
	GRIB: BOOL;
	LV_low_LK7: BOOL;
	LV_high_LK7: BOOL;
	LV_low_LK8: BOOL;
	LV_high_LK8: BOOL;
	LV_low_D2: BOOL;
	LV_high_D2: BOOL;
	stop_s: BOOL;
	pusk_LAN: BOOL;
	stop_LAN: BOOL;
	P: BOOL;
	err: BOOL;
END_VAR

VAR_OUTPUT
	ready: BOOL;
	KM: BOOL;
	work: BOOL;
	avar: BOOL;
END_VAR

VAR
	prom1: BOOL;
	sr_LK7: SR;
	low_LK7: BOOL;
	sr_LK8: SR;
	low_LK8: BOOL;
	sr_D2: SR;
	low_D2: BOOL;
END_VAR
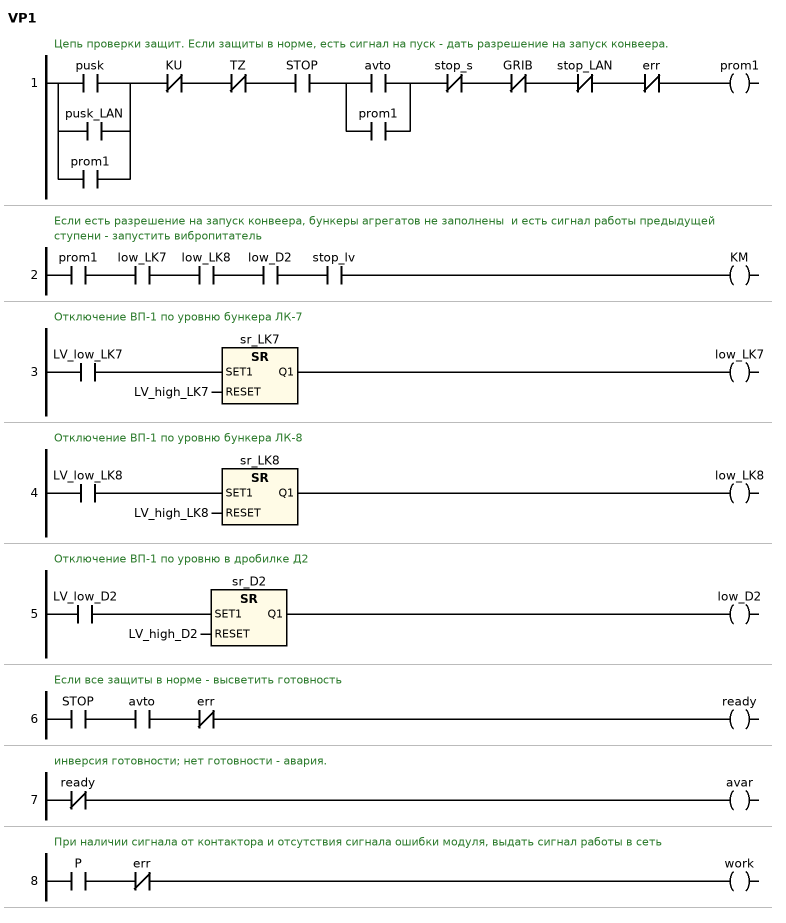
_LD_ (* Ladder Diagram *)
NETWORK 1 (* Цепь проверки защит. Если защиты в норме, есть сигнал на пуск - дать разрешение на запуск конвеера. *)
	{ [pusk] | [pusk_LAN] | [prom1] } - [/KU] - [/TZ] - [STOP] - { [avto] | [prom1] } - [/stop_s] - [/GRIB] - [/stop_LAN] - [/err] --- (prom1)
NETWORK 2 (* Если есть разрешение на запуск конвеера, бункеры агрегатов не заполнены  и есть сигнал работы предыдущей ступени - запустить вибропитатель *)
	[prom1] - [low_LK7] - [low_LK8] - [low_D2] - [stop_lv] --- (KM)
NETWORK 3 (* Отключение ВП-1 по уровню бункера ЛК-7 *)
	[LV_low_LK7] - sr_LK7:SR(SET1: *, RESET: LV_high_LK7) --- (low_LK7)
NETWORK 4 (* Отключение ВП-1 по уровню бункера ЛК-8 *)
	[LV_low_LK8] - sr_LK8:SR(SET1: *, RESET: LV_high_LK8) --- (low_LK8)
NETWORK 5 (* Отключение ВП-1 по уровню в дробилке Д2 *)
	[LV_low_D2] - sr_D2:SR(SET1: *, RESET: LV_high_D2) --- (low_D2)
NETWORK 6 (* Если все защиты в норме - высветить готовность *)
	[STOP] - [avto] - [/err] --- (ready)
NETWORK 7 (* инверсия готовности; нет готовности - авария. *)
	[/ready] --- (avar)
NETWORK 8 (* При наличии сигнала от контактора и отсутствия сигнала ошибки модуля, выдать сигнал работы в сеть *)
	[P] - [/err] --- (work)
_END_LD_
(* the same logic as Structured Text *)
(* Network 1: Цепь проверки защит. Если защиты в норме, есть сигнал на пуск - дать разрешение на запуск конвеера. *)
prom1 := (pusk OR pusk_LAN OR prom1) AND NOT KU AND NOT TZ AND STOP AND (avto OR prom1) AND NOT stop_s AND NOT GRIB AND NOT stop_LAN AND NOT err;
(* Network 2: Если есть разрешение на запуск конвеера, бункеры агрегатов не заполнены  и есть сигнал работы предыдущей ступени - запустить вибропитатель *)
KM := prom1 AND low_LK7 AND low_LK8 AND low_D2 AND stop_lv;
(* Network 3: Отключение ВП-1 по уровню бункера ЛК-7 *)
sr_LK7(SET1 := LV_low_LK7, RESET := LV_high_LK7);
low_LK7 := sr_LK7.Q1;
(* Network 4: Отключение ВП-1 по уровню бункера ЛК-8 *)
sr_LK8(SET1 := LV_low_LK8, RESET := LV_high_LK8);
low_LK8 := sr_LK8.Q1;
(* Network 5: Отключение ВП-1 по уровню в дробилке Д2 *)
sr_D2(SET1 := LV_low_D2, RESET := LV_high_D2);
low_D2 := sr_D2.Q1;
(* Network 6: Если все защиты в норме - высветить готовность *)
ready := STOP AND avto AND NOT err;
(* Network 7: инверсия готовности; нет готовности - авария. *)
avar := NOT ready;
(* Network 8: При наличии сигнала от контактора и отсутствия сигнала ошибки модуля, выдать сигнал работы в сеть *)
work := P AND NOT err;
END_FUNCTION_BLOCK

(* POU stop_VP1, LD *)
FUNCTION_BLOCK stop_VP1 (*блок управления включения/отключения агрегатов по уровню наполнения бункера*)
VAR_INPUT
	LV_in: REAL;
	LV_high_in: REAL;
	LV_low_in: REAL;
END_VAR
VAR_OUTPUT
	LV2_out: BOOL;
	LV1_out: BOOL;
END_VAR
VAR
	LV: WORD;
	LV_high: WORD;
	LV_low: WORD;

	LV_x10: REAL;
	LV_high_x10: REAL;
	LV_low_x10: REAL;

	ton1: TON;
	LV2: BOOL;
	lv_abs: REAL;
END_VAR
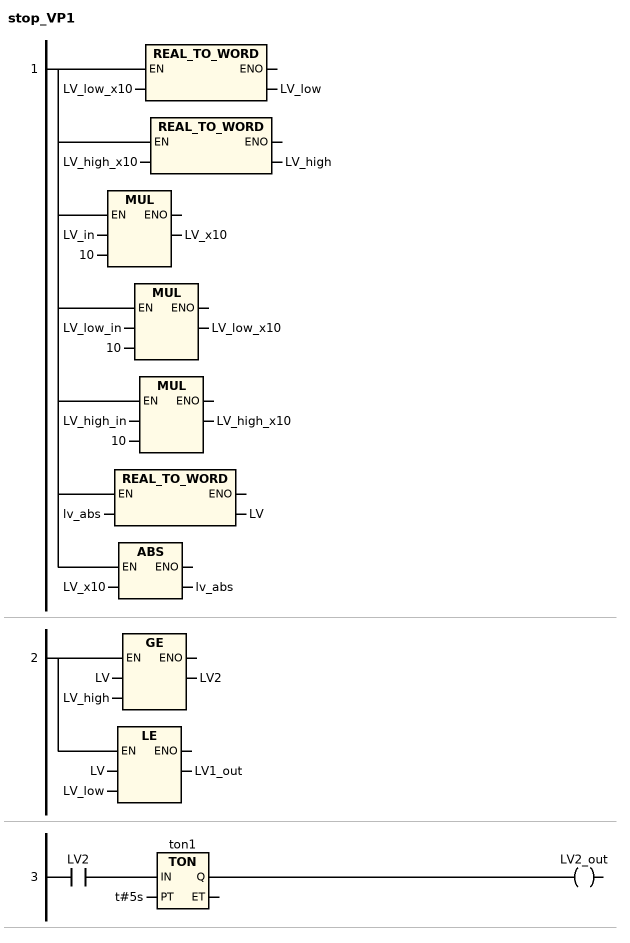
_LD_ (* Ladder Diagram *)
NETWORK 1
	*
		EN --- REAL_TO_WORD(LV_low_x10) => LV_low
		EN --- REAL_TO_WORD(LV_high_x10) => LV_high
		EN --- MUL(LV_in, 10) => LV_x10
		EN --- MUL(LV_low_in, 10) => LV_low_x10
		EN --- MUL(LV_high_in, 10) => LV_high_x10
		EN --- REAL_TO_WORD(lv_abs) => LV
		EN --- ABS(LV_x10) => lv_abs
NETWORK 2
	*
		EN --- GE(LV, LV_high) => LV2
		EN --- LE(LV, LV_low) => LV1_out
NETWORK 3
	[LV2] - ton1:TON(IN: *, PT: t#5s) --- (LV2_out)
_END_LD_
(* the same logic as Structured Text *)
(* Network 1 *)
LV_low := REAL_TO_WORD(LV_low_x10);
LV_high := REAL_TO_WORD(LV_high_x10);
LV_x10 := LV_in * 10;
LV_low_x10 := LV_low_in * 10;
LV_high_x10 := LV_high_in * 10;
LV := REAL_TO_WORD(lv_abs);
lv_abs := ABS(LV_x10);
(* Network 2 *)
LV2 := LV >= LV_high;
LV1_out := LV <= LV_low;
(* Network 3 *)
ton1(IN := LV2, PT := t#5s);
LV2_out := ton1.Q;
END_FUNCTION_BLOCK

(* POU signals, CFC *)
FUNCTION_BLOCK signals
VAR_INPUT
	KU_D2_in: BOOL;
	RMS2_2_in: BOOL;
	avto_D2_in: BOOL;
	work_D2_in: BOOL;
	ready_D2_in: BOOL;
	TZD2_in: BOOL;

	KU_D3_in: BOOL;
	TZN_D3_in: BOOL;
	UM_D3_in: BOOL;
	KPM_D3_in: BOOL;
	TZV_D3_in: BOOL;
	avto_D3_in: BOOL;
	KUD3_D3_in: BOOL;
	TZD3_D3_in: BOOL;
	work_D3_in: BOOL;
	ready_D3_in: BOOL;
	TM_D3_in: BOOL;
	RMS_D3_in: BOOL;
	DM_D3_in: BOOL;

	KU_D4_in: BOOL;
	TZN_D4_in: BOOL;
	UM_D4_in: BOOL;
	KPM_D4_in: BOOL;
	TZV_D4_in: BOOL;
	avto_D4_in: BOOL;
	KUD3_D4_in: BOOL;
	TZD3_D4_in: BOOL;
	work_D4_in: BOOL;
	ready_D4_in: BOOL;
	TM_D4_in: BOOL;
	RMS_D4_in: BOOL;
	DM_D4_in: BOOL;

	KU_LK10_in: BOOL;
	TZ_LK10_in: BOOL;
	tros_LK10_in: BOOL;
	shod_LK10_in: BOOL;
	ogr_LK10_in: BOOL;
	avto_LK10_in: BOOL;
	ready_LK10_in: BOOL;
	work_LK10_in: BOOL;

	KU_LK11_in: BOOL;
	TZ_LK11_in: BOOL;
	tros_LK11_in: BOOL;
	shod_LK11_in: BOOL;
	ogr_LK11_in: BOOL;
	avto_LK11_in: BOOL;
	ready_LK11_in: BOOL;
	work_LK11_in: BOOL;

	KU_LK12_in: BOOL;
	TZ_LK12_in: BOOL;
	tros_LK12_in: BOOL;
	shod_LK12_in: BOOL;
	ogr_LK12_in: BOOL;
	avto_LK12_in: BOOL;
	ready_LK12_in: BOOL;
	work_LK12_in: BOOL;

	KU_LK13_in: BOOL;
	TZ_LK13_in: BOOL;
	tros_LK13_in: BOOL;
	shod_LK13_in: BOOL;
	ogr_LK13_in: BOOL;
	avto_LK13_in: BOOL;
	ready_LK13_in: BOOL;
	work_LK13_in: BOOL;

	avto_GR3_in: BOOL;
	KU_GR3_in: BOOL;
	TZ_GR3_in: BOOL;
	ready_GR3_in: BOOL;
	work_GR3_in: BOOL;
	STOP_GR3_in: BOOL;

	KU_LK7_in: BOOL;
	TZ_LK7_in: BOOL;
	tros_LK7_in: BOOL;
	shod_LK7_in: BOOL;
	ogr_LK7_in: BOOL;
	avto_LK7_in: BOOL;
	ready_LK7_in: BOOL;
	work_LK7_in: BOOL;

	KU_LK8_in: BOOL;
	TZ_LK8_in: BOOL;
	tros_LK8_in: BOOL;
	shod_LK8_in: BOOL;
	ogr_LK8_in: BOOL;
	avto_LK8_in: BOOL;
	ready_LK8_in: BOOL;
	work_LK8_in: BOOL;

	KU_LK6_in: BOOL;
	TZ_LK6_in: BOOL;
	tros_LK6_in: BOOL;
	shod_LK6_in: BOOL;
	ogr_LK6_in: BOOL;
	avto_LK6_in: BOOL;
	ready_LK6_in: BOOL;
	work_LK6_in: BOOL;

	KU_LK9_in: BOOL;
	TZ_LK9_in: BOOL;
	tros_LK9_in: BOOL;
	ogr_LK9_in: BOOL;
	shod_LK9_in: BOOL;
	avto_LK9_in: BOOL;
	ready_LK9_in: BOOL;
	work_LK9_in: BOOL;

	KU_LP1_3_in: BOOL;
	in_020_in: BOOL;
	in_040_in: BOOL;
	in_020_4070_in: BOOL;
	TZ1_LP1_3_in: BOOL;
	TZ2_LP1_3_in: BOOL;
	TZ3_LP1_3_in: BOOL;
	PRO_LP1_3_in: BOOL;
	avto_LP1_3_in: BOOL;
	ready_LP1_3_in: BOOL;
	work_LP1_3_in: BOOL;
	stop2_LP1_3_in: BOOL;

	avto_GR2_in: BOOL;
	KU_GR2_in: BOOL;
	TZ_GR2_in: BOOL;
	ready_GR2_in: BOOL;
	work_GR2_in: BOOL;
	STOP_GR2_in: BOOL;

	KU_LK5_in: BOOL;
	TZ_LK5_in: BOOL;
	tros_LK5_in: BOOL;
	shod_LK5_in: BOOL;
	ogr_LK5_in: BOOL;
	avto_LK5_in: BOOL;
	ready_LK5_in: BOOL;
	work_LK5_in: BOOL;

	KU_LK4_in: BOOL;
	TZ_LK4_in: BOOL;
	tros_LK4_in: BOOL;
	shod_LK4_in: BOOL;
	avto_LK4_in: BOOL;
	ready_LK4_in: BOOL;
	work_LK4_in: BOOL;
	MD3_LK4_in: BOOL;

	avto_GR1_in: BOOL;
	KU_GR1_in: BOOL;
	TZ_GR1_in: BOOL;
	ready_GR1_in: BOOL;
	work_GR1_in: BOOL;
	STOP_GR1_in: BOOL;

	KU_LK2_in: BOOL;
	TZ_LK2_in: BOOL;
	tros_LK2_in: BOOL;
	shod_LK2_in: BOOL;
	ogr_LK2_in: BOOL;
	avto_LK2_in: BOOL;
	ready_LK2_in: BOOL;
	work_LK2_in: BOOL;

	KU_LK3_in: BOOL;
	TZ_LK3_in: BOOL;
	tros_LK3_in: BOOL;
	shod_LK3_in: BOOL;
	ogr_LK3_in: BOOL;
	avto_LK3_in: BOOL;
	ready_LK3_in: BOOL;
	work_LK3_in: BOOL;

	avto_LP4_in: BOOL;
	ready_LP4_in: BOOL;
	work_LP4_in: BOOL;
	MD2_LP4_in: BOOL;

	avto_LP5_in: BOOL;
	ready_LP5_in: BOOL;
	work_LP5_in: BOOL;
	STOP_LP5_in: BOOL;
	output_Hz_LP5_in: WORD;
	MD2_LP5_in: BOOL;

	avto_VP1_in: BOOL;
	ready_VP1_in: BOOL;
	work_VP1_in: BOOL;
	STOP_VP1_in: BOOL;
	KU_VP1_in: BOOL;
	TZ_VP1_in: BOOL;

	avto_all_in: BOOL;
	pusk_in: BOOL;

	PP1_in: BOOL;

	LV_GR1_in: REAL;
	LV_LK7_in: REAL;
	LV_LK8_in: REAL;
	LV_D2_in: REAL;

	lev_up_cyc_in: BOOL;
	pre_cyc_in: BOOL;
	ku_cyc_in: BOOL;
	tz_cyc_in: BOOL;
	ready_cyc_in: BOOL;
	work_cyc_in: BOOL;
	shnek_up_cyc_in: BOOL;
	avar_cyc_in: BOOL;
	gribok_in: BOOL;
	TM_D3_word_in: WORD;
	TM_D4_word_in: WORD;
	avar_FC_lp5_in: BOOL;
	lev_down_cyc_in: BOOL;
END_VAR
VAR_OUTPUT
	KU_D2_out: BOOL;
	RMS2_2_out: BOOL;
	avto_D2_out: BOOL;
	work_D2_out: BOOL;
	ready_D2_out: BOOL;
	TZD2_out: BOOL;

	KU_D3_out: BOOL;
	TZN_D3_out: BOOL;
	UM_D3_out: BOOL;
	KPM_D3_out: BOOL;
	TZV_D3_out: BOOL;
	avto_D3_out: BOOL;
	KUD3_D3_out: BOOL;
	TZD3_D3_out: BOOL;
	work_D3_out: BOOL;
	ready_D3_out: BOOL;
	TM_D3_out: BOOL;
	RMS_D3_out: BOOL;
	DM_D3_out: BOOL;

	KU_D4_out: BOOL;
	TZN_D4_out: BOOL;
	UM_D4_out: BOOL;
	KPM_D4_out:BOOL;
	TZV_D4_out: BOOL;
	KUD3_D4_out: BOOL;
	TZD3_D4_out: BOOL;
	work_D4_out:BOOL;
	ready_D4_out: BOOL;
	avto_D4_out: BOOL;
	TM_D4_out: BOOL;
	RMS_D4_out: BOOL;
	DM_D4_out: BOOL;

	KU_LK10_out: BOOL;
	TZ_LK10_out: BOOL;
	tros_LK10_out: BOOL;
	shod_LK10_out: BOOL;
	ogr_LK10_out: BOOL;
	avto_LK10_out: BOOL;
	ready_LK10_out: BOOL;
	work_LK10_out: BOOL;

	KU_LK11_out: BOOL;
	TZ_LK11_out: BOOL;
	tros_LK11_out: BOOL;
	shod_LK11_out: BOOL;
	ogr_LK11_out: BOOL;
	avto_LK11_out: BOOL;
	ready_LK11_out: BOOL;
	work_LK11_out: BOOL;

	KU_LK12_out: BOOL;
	TZ_LK12_out: BOOL;
	tros_LK12_out: BOOL;
	shod_LK12_out: BOOL;
	ogr_LK12_out: BOOL;
	avto_LK12_out: BOOL;
	ready_LK12_out: BOOL;
	work_LK12_out: BOOL;

	KU_LK13_out: BOOL;
	TZ_LK13_out: BOOL;
	tros_LK13_out: BOOL;
	shod_LK13_out: BOOL;
	ogr_LK13_out: BOOL;
	avto_LK13_out: BOOL;
	ready_LK13_out: BOOL;
	work_LK13_out: BOOL;

	avto_GR3_out: BOOL;
	KU_GR3_out: BOOL;
	TZ_GR3_out: BOOL;
	ready_GR3_out: BOOL;
	work_GR3_out: BOOL;
	STOP_GR3_out: BOOL;

	KU_LK7_out: BOOL;
	TZ_LK7_out: BOOL;
	tros_LK7_out: BOOL;
	shod_LK7_out: BOOL;
	ogr_LK7_out: BOOL;
	avto_LK7_out: BOOL;
	ready_LK7_out: BOOL;
	work_LK7_out: BOOL;

	KU_LK8_out: BOOL;
	TZ_LK8_out: BOOL;
	tros_LK8_out: BOOL;
	shod_LK8_out: BOOL;
	ogr_LK8_out: BOOL;
	avto_LK8_out: BOOL;
	ready_LK8_out: BOOL;
	work_LK8_out: BOOL;

	KU_LK6_out: BOOL;
	TZ_LK6_out: BOOL;
	tros_LK6_out: BOOL;
	shod_LK6_out: BOOL;
	ogr_LK6_out: BOOL;
	avto_LK6_out: BOOL;
	ready_LK6_out: BOOL;
	work_LK6_out: BOOL;

	KU_LK9_out: BOOL;
	TZ_LK9_out: BOOL;
	tros_LK9_out: BOOL;
	shod_LK9_out: BOOL;
	ogr_LK9_out: BOOL;
	avto_LK9_out: BOOL;
	ready_LK9_out: BOOL;
	work_LK9_out: BOOL;

	KU_LP1_3_out: BOOL;
	in_020_out: BOOL;
	in_040_out: BOOL;
	in_020_4070_out: BOOL;
	TZ1_LP1_3_out: BOOL;
	TZ2_LP1_3_out: BOOL;
	TZ3_LP1_3_out: BOOL;
	PRO_LP1_3_out: BOOL;
	avto_LP1_3_out: BOOL;
	ready_LP1_3_out: BOOL;
	work_LP1_3_out: BOOL;
	stop2_LP1_3_out: BOOL;

	avto_GR2_out: BOOL;
	KU_GR2_out: BOOL;
	TZ_GR2_out: BOOL;
	ready_GR2_out: BOOL;
	work_GR2_out: BOOL;
	STOP_GR2_out: BOOL;

	KU_LK5_out: BOOL;
	TZ_LK5_out: BOOL;
	tros_LK5_out: BOOL;
	shod_LK5_out: BOOL;
	ogr_LK5_out: BOOL;
	avto_LK5_out: BOOL;
	ready_LK5_out: BOOL;
	work_LK5_out: BOOL;

	KU_LK4_out: BOOL;
	TZ_LK4_out: BOOL;
	tros_LK4_out: BOOL;
	shod_LK4_out: BOOL;
	avto_LK4_out: BOOL;
	ready_LK4_out: BOOL;
	work_LK4_out: BOOL;
	MD3_LK4_out: BOOL;

	avto_GR1_out: BOOL;
	KU_GR1_out: BOOL;
	TZ_GR1_out: BOOL;
	ready_GR1_out: BOOL;
	work_GR1_out: BOOL;
	STOP_GR1_out: BOOL;

	KU_LK2_out: BOOL;
	TZ_LK2_out: BOOL;
	tros_LK2_out: BOOL;
	shod_LK2_out: BOOL;
	ogr_LK2_out: BOOL;
	avto_LK2_out: BOOL;
	ready_LK2_out: BOOL;
	work_LK2_out: BOOL;

	KU_LK3_out: BOOL;
	TZ_LK3_out: BOOL;
	tros_LK3_out: BOOL;
	shod_LK3_out: BOOL;
	ogr_LK3_out: BOOL;
	avto_LK3_out: BOOL;
	ready_LK3_out: BOOL;
	work_LK3_out: BOOL;

	avto_LP4_out: BOOL;
	ready_LP4_out: BOOL;
	work_LP4_out: BOOL;
	MD2_LP4_out: BOOL;
	output_Hz_LP4_out: WORD;

	avto_LP5_out: BOOL;
	ready_LP5_out: BOOL;
	work_LP5_out: BOOL;
	STOP_LP5_out: BOOL;
	MD2_LP5_out: BOOL;
	output_Hz_LP5_out: WORD;

	avto_VP1_out: BOOL;
	ready_VP1_out: BOOL;
	work_VP1_out: BOOL;
	STOP_VP1_out: BOOL;
	KU_VP1_out: BOOL;
	TZ_VP1_out: BOOL;

	avto_all_out: BOOL;
	pusk_out: BOOL;

	PP1_out: BOOL;

	LV_GR1_out: WORD;
	LV_LK7_out: WORD;
	LV_LK8_out: WORD;
	LV_D2_out: WORD;

	lev_up_cyc_out: BOOL;
	pre_cyc_out: BOOL;
	ku_cyc_out: BOOL;
	tz_cyc_out: BOOL;
	ready_cyc_out: BOOL;
	work_cyc_out: BOOL;
	shnek_up_cyc_out: BOOL;
	avar_cyc_out: BOOL;
	gribok_out: BOOL;
	TM_D3_word_out: WORD;
	TM_D4_word_out: WORD;
	avar_FC_lp5_out: BOOL;
	lev_down_cyc_out: BOOL;
END_VAR
VAR
	LV_LK7_prom: WORD;
	LV_LK8_prom: WORD;
	LV_GR1_prom: WORD;
	LV_D2_prom: WORD;
	LV_LK7_x10: REAL;
	LV_LK8_x10: REAL;
	LV_GR1_x10: REAL;
	LV_D2_x10: REAL;
END_VAR
